(* CoDeSys 2.3.9.41 project: KS Babaevskaya.pro *)
(* Libraries: PID_Regulators.lib 28.12.06 17:47:54, SysLibTime.lib 20.2.06 13:31:16, Util.lib 18.5.10 15:14:28, STANDARD.LIB 4.10.05 11:14:46, IECSFC.LIB 13.4.06 15:51:28, ANALYZATION.LIB 5.10.99 09:05:06 *)

(* PLC configuration (modules and I/O channels)
Fast discrete inputs [I_SIMPLE_INPUT] node 0, in %IB0 out %QB0 {Filtrationtime = 10}
  DD1_DI0 AT %IX0.0 [BitInput] резерв
  DD1_DI1 AT %IX0.1 [BitInput] резерв
  DD1_DI2 AT %IX0.2 [BitInput] резерв
  DD1_DI3 AT %IX0.3 [BitInput] резерв
Discrete inputs [ID130] node 1, in %IB1 out %QB1 {Filtrationtime_GeneralINP = 10; Visibility = No; PinCount = 12}
  AT %IB1.0 [ByteInput] 8 discrete inputs
  AT %IB1.1 [ByteInput] 4 discrete inputs
Discrete outputs [ID131] node 2, in %IB2 out %QB2 {SafeValueByte = 0; SafeValueByteM = 0; Visibility = No; PinCount = 12}
  AT %QB2.0 [ByteOutput] 8 discrete outputs
  AT %QB2.1 [ByteOutput] 4 discrete outputs
ID125	50Hz 2Por	50Hz 2PorBYTEFast analog i AT %IR3.0 [FloatInputP] putsIB%QB%MB%	MDD1_AI0&AI #1 - датчик температуры в помещении {AIN_TYPE = 4-20 mA; Peak_Filtr = 200; Flt_Ch = Off; TauRC = 10; MinFV = 0; MaxFV = 100}
DD1_AI1 AT %IR3.1 [FloatInputP] AI #2 - расходомер FT01.01 (на входе, до отстойника) {AIN_TYPE = 4-20 mA; Peak_Filtr = 200; Flt_Ch = Off; TauRC = 10; MinFV = 0; MaxFV = 600}
DD1_AI2 AT %IR3.2 [FloatInputP] AI #3 - расходомер FT01.02 (на выходе, после отстойника) {AIN_TYPE = 4-20 mA; Peak_Filtr = 200; Flt_Ch = Off; TauRC = 10; MinFV = 0; MaxFV = 600}
DD1_AI3 AT %IR3.3 [FloatInputP] AI #4 - рН-метр QE01.01 (на входе, до отстойника) {AIN_TYPE = 4-20 mA; Peak_Filtr = 200; Flt_Ch = Off; TauRC = 10; MinFV = 0; MaxFV = 20000.0}
DD1_AI4 AT %IR3.4 [FloatInputP] AI #5 - рН-метр QE01.02 (на выходе, после отстойника) {AIN_TYPE = 4-20 mA; Peak_Filtr = 200; Flt_Ch = Off; TauRC = 10; MinFV = 0; MaxFV = 20000.0}
DD1_AI5 AT %IR3.5 [FloatInputP] AI #6 - сигнал от ФПК, давление на входе {AIN_TYPE = 4-20 mA; Peak_Filtr = 200; Flt_Ch = Off; TauRC = 10; MinFV = 0; MaxFV = 20000.0}
DD1_AI6 AT %IR3.6 [FloatInputP] AI #7 - резерв {AIN_TYPE = 4-20 mA; Peak_Filtr = 200; Flt_Ch = Off; TauRC = 10; MinFV = 0; MaxFV = 20000.0}
DD1_AI7 AT %IR3.7 [FloatInputP] AI #8 - обратная связь от ЧРП Н01.05 (частота, обороты, или ток) {AIN_TYPE = 4-20 mA; Peak_Filtr = 200; Flt_Ch = Off; TauRC = 10; MinFV = 0; MaxFV = 20000.0}
AT %IW3.8 [WordInput] AI read time (10ms)
Analog outputs [ID126] node 4, in %IB4 out %QB4
  DD1_AO0 AT %QR4.0 [FloatOutputP] AO #1 - управление ЧРП Н01.05 (поддержание расхода по расходомеру FT01.02) {AOUT_TYPE = 4-20 mA; SafeValueREAL = 0.0}
  DD1_AO1 AT %QR4.1 [FloatOutputP] AO #2 - управление ЧРП НД08.03/01 (подача флокулянта на входе, до отстойника, по FT01.01) {AOUT_TYPE = 4-20 mA; SafeValueREAL = 0.0}
  DD1_AO2 AT %QR4.2 [FloatOutputP] AO #3 - управление ЧРП НД08.03/02 (подача флокулянта на входе, до отстойника, по FT01.01) {AOUT_TYPE = 4-20 mA; SafeValueREAL = 0.0}
  DD1_AO3 AT %QR4.3 [FloatOutputP] AO #4 - управление НД05.02/01 (подача 10%NaCl из УПГ на входе, до отстойника, по FT01.01) {AOUT_TYPE = 4-20 mA; SafeValueREAL = 0.0}
Special input [ID103] node 5, in %IB5 out %QB5 {Filtrationtime = 1000; PinCount = 1; WatchDogPeriod = 400; PollPeriod = 3000; Visibility = No}
  AT %IX5.0 [BitInput] Special input
Special output [ID104] node 6, in %IB6 out %QB6 {Visibility = No; PinCount = 1}
  AT %QX6.0 [BitOutput] Special output
AT %QD7.0 [DWordOutput] Last address
AT %QW7.1 [WordOutput] Last error
RS-485-1 [COM1_USART] node 0, in %IB7.0 out %QB7.0 {CommunicationSpeed = 57600; Parity = NO PARITY CHECK; BitLength = 8 bits; StopLength = One stop bit; InterfaceType = RS485; FrameOriented = RTU; Timeout = 0; Visibility = No}
Universal Modbus device [ID2000] node 1, in %IB7.1 out %QB7.1 {ModuleIP = 10:0:0:102; ServiceTimeout = 20; TCPport = 502; NetMode = Serial; ModuleSlaveAddress = 2; RequestType = Both; PeriodOfService = 100; Visibility = No; RepeatCounter = 0; ByteSequence = Trace_mode}
  AT %QB7.1.0 [ComChannel] Command (0xff - Start)
DD2_DO AT %QD7.1.0.0 [DWordOutput] регистр 0, команда 0х0f
Universal Modbus device [ID2000] node 2, in %IB7.2 out %QB7.2 {ModuleIP = 10:0:0:103; ServiceTimeout = 20; TCPport = 502; NetMode = Serial; ModuleSlaveAddress = 3; RequestType = Both; PeriodOfService = 100; Visibility = No; RepeatCounter = 0; ByteSequence = Trace_mode}
  AT %QB7.2.0 [ComChannel] Command (0xff - Start)
DD3_DO AT %QD7.2.0.0 [DWordOutput]
Universal Modbus device [ID2000] node 3, in %IB7.3 out %QB7.3 {ModuleIP = 10:0:0:104; ServiceTimeout = 20; TCPport = 502; NetMode = Serial; ModuleSlaveAddress = 4; RequestType = Both; PeriodOfService = 100; Visibility = No; RepeatCounter = 0; ByteSequence = Trace_mode}
  AT %QB7.3.0 [ComChannel] Command (0xff - Start)
DD4_DO AT %QD7.3.0.0 [DWordOutput]
Universal Modbus device [ID2000] node 4, in %IB7.4 out %QB7.4 {ModuleIP = 10:0:0:105; ServiceTimeout = 20; TCPport = 502; NetMode = Serial; ModuleSlaveAddress = 5; RequestType = Both; PeriodOfService = 100; Visibility = No; RepeatCounter = 0; ByteSequence = Trace_mode}
  AT %QB7.4.0 [ComChannel] Command (0xff - Start)
DD5_DI AT %ID7.4.0.0 [DWordInput]
Universal Modbus device [ID2000] node 5, in %IB7.5 out %QB7.5 {ModuleIP = 10:0:0:106; ServiceTimeout = 20; TCPport = 502; NetMode = Serial; ModuleSlaveAddress = 6; RequestType = Both; PeriodOfService = 100; Visibility = No; RepeatCounter = 0; ByteSequence = Trace_mode}
  AT %QB7.5.0 [ComChannel] Command (0xff - Start)
DD6_DI AT %ID7.5.0.0 [DWordInput]
Universal Modbus device [ID2000] node 6, in %IB7.6 out %QB7.6 {ModuleIP = 10:0:0:107; ServiceTimeout = 20; TCPport = 502; NetMode = Serial; ModuleSlaveAddress = 7; RequestType = Both; PeriodOfService = 100; Visibility = No; RepeatCounter = 0; ByteSequence = Trace_mode}
  AT %QB7.6.0 [ComChannel] Command (0xff - Start)
DD7_DI AT %ID7.6.0.0 [DWordInput]
Universal Modbus device [ID2000] node 7, in %IB7.7 out %QB7.7 {ModuleIP = 10:0:0:108; ServiceTimeout = 20; TCPport = 502; NetMode = Serial; ModuleSlaveAddress = 8; RequestType = Both; PeriodOfService = 100; Visibility = No; RepeatCounter = 0; ByteSequence = Trace_mode}
  AT %QB7.7.0 [ComChannel] Command (0xff - Start)
DD8_DI AT %ID7.7.0.0 [DWordInput]
Universal Modbus device [ID2000] node 8, in %IB7.8 out %QB7.8 {ModuleIP = 10:0:0:109; ServiceTimeout = 20; TCPport = 502; NetMode = Serial; ModuleSlaveAddress = 9; RequestType = Both; PeriodOfService = 100; Visibility = No; RepeatCounter = 0; ByteSequence = Trace_mode}
  AT %QB7.8.0 [ComChannel] Command (0xff - Start)
DD9_DI AT %ID7.8.0.0 [DWordInput]
Universal Modbus device [ID2000] node 9, in %IB7.9 out %QB7.9 {ModuleIP = 10:0:0:110; ServiceTimeout = 20; TCPport = 502; NetMode = Serial; ModuleSlaveAddress = 10; RequestType = Both; PeriodOfService = 100; Visibility = No; RepeatCounter = 0; ByteSequence = Trace_mode}
  AT %QB7.9.0 [ComChannel] Command (0xff - Start)
DD10_AO0 AT %QW7.9.0.0 [WordOutput]
DD10_AO1 AT %QW7.9.1.0 [WordOutput]
DD10_AO2 AT %QW7.9.2.0 [WordOutput]
DD10_AO3 AT %QW7.9.3.0 [WordOutput]
DD10_AO4 AT %QW7.9.4.0 [WordOutput]
DD10_AO5 AT %QW7.9.5.0 [WordOutput]
DD10_AO6 AT %QW7.9.6.0 [WordOutput]
DD10_AO7 AT %QW7.9.7.0 [WordOutput]
*)

(* POU PLC_PRG, CFC *)
PROGRAM PLC_PRG
VAR
	temperatureLimits: LIMITALARM;		(*блок контроля границ допустимой температуры в помещении*)
	minTemperature: BYTE;		(*температура, ниже которой будет подан сигнал НИЗКАЯ ТЕМПЕРАТУРА*)
	maxTemperature: BYTE;		(*Температура, выше которой будет подан сигнал ВЫСОКАЯ ТЕМПЕРАТУРА*)
	alarmHighTemperature: BOOL;		(*температура выше заданного диапазона*)
	alarmLowTemperature: BOOL;		(*температура ниже заданного диапазона*)
	temperatureValue: REAL;		(*значение температуры в помещении*)
	DD1_AI0_temperature: DECODE_FLOAT;		(*блок контроля состояния аналогового входа ПЛК для датчика температуры в помещении*)
	DD1_AI1_flow: DECODE_FLOAT;		(*блок контроля состояния аналогового входа ПЛК для расходомера FT01.01*)
	DD1_AI1_error: BOOL;		(*авария входа AI2 (возможно, обрыв)*)
	DD1_AI0_error: BOOL;		(*авария входа AI1 (возможно, обрыв)*)


	tempCTU1: CTU;
	tempStartAuto: BOOL;
	tempReset1: BOOL;
	tempReset2: BOOL;
	tempPV: WORD := 15;		(*по умолчанию = 15*)
	tempCTU2: CTU;
	tempStartPump1: BOOL;
	tempStartPump2: BOOL;
	counterPump1: WORD;
	counterPump2: WORD;
	tempErrorPump1: BOOL;
	tempErrorPump2: BOOL;
	tempStopPump1: BOOL;
	tempStopPump2: BOOL;
	tempFtrigPump1: F_TRIG;
	tempRtrigPump1: R_TRIG;
	tempRSpump1: RS;
	tempStartStopPump1: BOOL;
	tempStartStopPump2: BOOL;
	tempPump1ON: BOOL;
	tempPump2ON: BOOL;
	tempRtrigPump2: R_TRIG;
	tempFtrigPump2: F_TRIG;
	tempRSpump2: RS;
	errorPump1Trig: RS;
	tempAlarmReset: BOOL;
	errorPump2Trig: RS;
	tempPump1EmergencyON: BOOL;
	tempPump1NormalON: BOOL;
	tempPump2NormalON: BOOL;
	tempPump2EmergencyON: BOOL;
	tempMan2Pump: ManualTwoPumpManager;
	tempalarmPump1: BOOL;
	tempalarmPump2: BOOL;
	tempalarmPump1RStrig: RS;
	tempalarmPump2RStrig: RS;
	alarmReset: BOOL;
	startStopPump1: BOOL;
	pump2ON: BOOL;
	alarmPump1: BOOL;
	startStopPump2: BOOL;
	pump1ON: BOOL;
	alarmPump2: BOOL;
	alarmPump2RStrig: RS;
	pump1EmergencyON: BOOL;
	pump2NormalON: BOOL;
	pump2EmergencyON: BOOL;
	RSpump2: RS;
	RtrigPump2: R_TRIG;
	FtrigPump2: F_TRIG;
	alarmPump1RStrig: RS;
	pump1NormalON: BOOL;
	RSpump1: RS;
	FtrigPump1: F_TRIG;
	RtrigPump1: R_TRIG;
	counterStart: BOOL;
	counterPump1ON: BOOL;
	counterPump2ON: BOOL;
	tempRtrig: R_TRIG;
	tempFtrig: F_TRIG;
	tempRStrig: RS;
	tempSRtrig2: SR;
	tempSRtrig1: SR;
	tempRStrig1: RS;
	tempRStrig2: RS;
	tempValueToResetCTU: WORD;
	tempCTU1reset: BOOL;
	tempCTU2reset: BOOL;
	tempCounterStart: BOOL;
	tempCounterPump1: WORD;
	tempCounterPump2: WORD;
	tempCounterTwoPumpManager: CounterTwoPumpManager;
	tempTON1: TON;
	tempBLINK: BLINK;
	tempRTC: RTC;
	tempCTU21: CTU;
	tempTIMEcdt: DT;
	tempTIMEPDT: DT;
	tempCTU22: CTU;
	tempSema1: SEMA;
	tempFTrig21: F_TRIG;
	tempTIME: TIME;
	tempTimeBlink: TIME;
	tempTIMEboolQ: BOOL;
	workTimePump1ON: BOOL;
	workTimePump2ON: BOOL;
	tempTIME2: TIME;
	tempRTrig23: R_TRIG;
	tempRStrig24: RS;
	tempRStrigTIME2: RS;
	tempRStrigTIME: RS;
	tempTOF1: TOF;
	tempTP1: TP;
	tempRStrig23: RS;
	tempRTrig21: R_TRIG;
	tempVARtime: DWORD;
	tempRStrig11: RS;
	tempRStrig12: RS;
	tempFtrig22: F_TRIG;
	tempFTrig24: F_TRIG;
	tempFTrig25: F_TRIG;
	currentWorkTimePump1: TIME;
	currentWorkTimePump2: TIME;
	tempTwoPumpFullManager: TwoPumpManager;
	tempWorkTimeStart: BOOL;
	pump1Time: TIME;
	pump2Time: TIME;
	tempWorkTimeReset: BOOL;
END_VAR
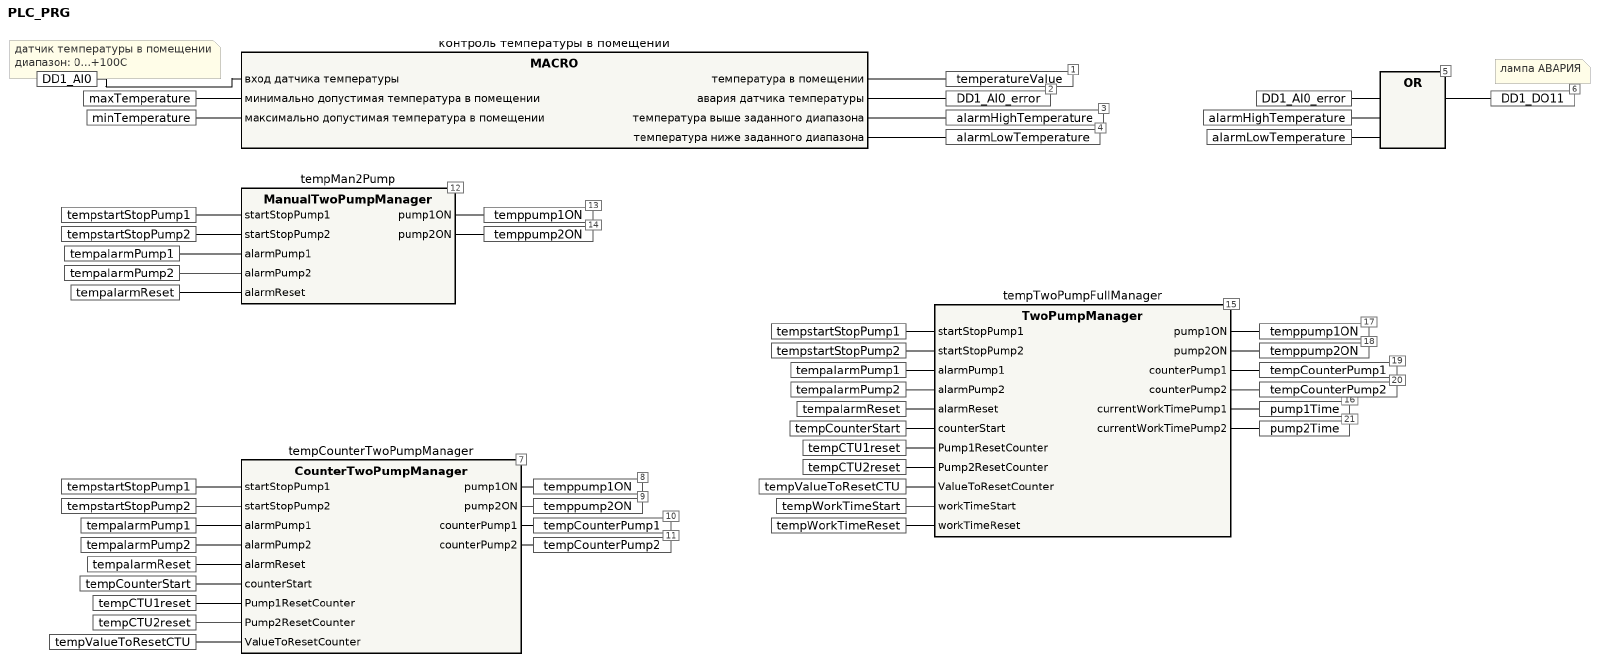
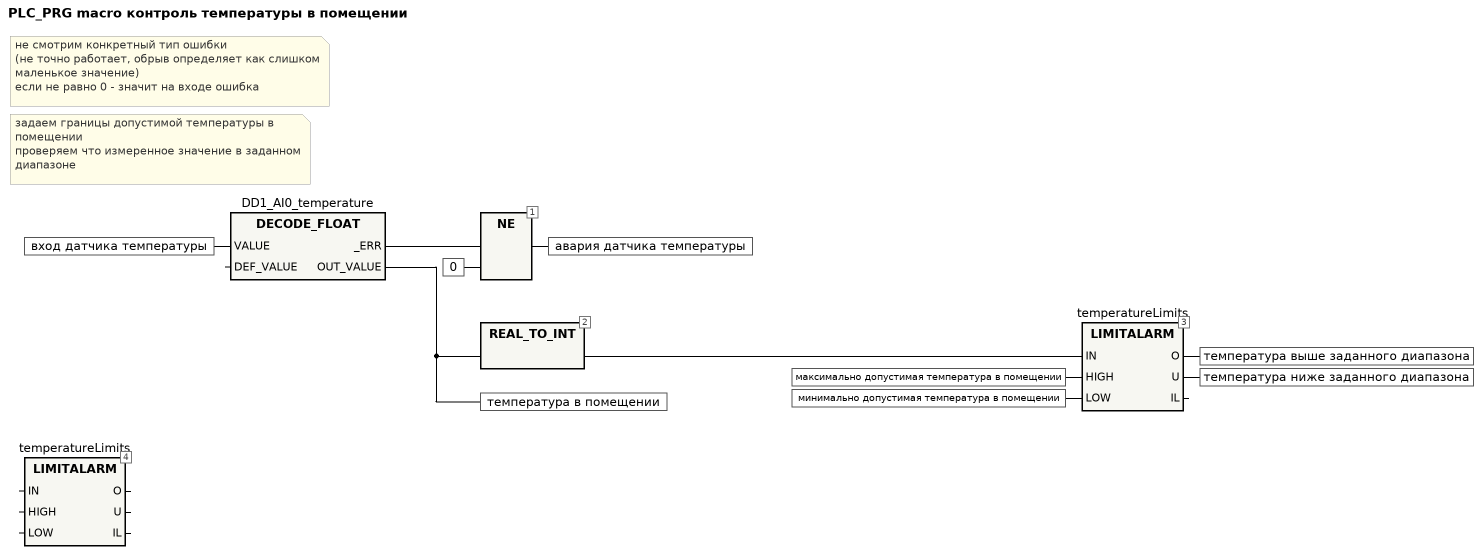
_CFC_ (* Continuous Function Chart, elements in execution order *)
(* датчик температуры в помещении / диапазон: 0...+100С *)
(* лампа АВАРИЯ *)
#0 MACRO контроль температуры в помещении(pin 1 "вход датчика температуры": DD1_AI0, pin 2 "минимально допустимая температура в помещении": maxTemperature, pin 3 "максимально допустимая температура в помещении": minTemperature)
	(* не смотрим конкретный тип ошибки / (не точно работает, обрыв определяет как слишком маленькое значение) / если не равно 0 - значит на входе ошибка *)
	(* задаем границы допустимой температуры в помещении / проверяем что измеренное значение в заданном диапазоне *)
	#1 DD1_AI0_temperature:DECODE_FLOAT(VALUE: pin 1, DEF_VALUE: -)
	#2 NE(#1._ERR, 0)
	out 2 "авария датчика температуры" <= #2
	out 1 "температура в помещении" <= #1.OUT_VALUE
	#3 REAL_TO_INT(#1.OUT_VALUE)
	#4 temperatureLimits:LIMITALARM(IN: #3, HIGH: pin 3, LOW: pin 2)
	out 3 "температура выше заданного диапазона" <= #4.O
	out 4 "температура ниже заданного диапазона" <= #4.U
	#5 temperatureLimits:LIMITALARM(IN: -, HIGH: -, LOW: -)
END_MACRO
#6 temperatureValue <= #0.out 1
#7 DD1_AI0_error <= #0.out 2
#8 alarmHighTemperature <= #0.out 3
#9 alarmLowTemperature <= #0.out 4
#10 OR(DD1_AI0_error, alarmHighTemperature, alarmLowTemperature)
#11 DD1_DO11 <= #10
#12 tempCounterTwoPumpManager:CounterTwoPumpManager(startStopPump1: tempstartStopPump1, startStopPump2: tempstartStopPump2, alarmPump1: tempalarmPump1, alarmPump2: tempalarmPump2, alarmReset: tempalarmReset, counterStart: tempCounterStart, Pump1ResetCounter: tempCTU1reset, Pump2ResetCounter: tempCTU2reset, ValueToResetCounter: tempValueToResetCTU)
#13 temppump1ON <= #12.pump1ON
#14 temppump2ON <= #12.pump2ON
#15 tempCounterPump1 <= #12.counterPump1
#16 tempCounterPump2 <= #12.counterPump2
#17 tempMan2Pump:ManualTwoPumpManager(startStopPump1: tempstartStopPump1, startStopPump2: tempstartStopPump2, alarmPump1: tempalarmPump1, alarmPump2: tempalarmPump2, alarmReset: tempalarmReset)
#18 temppump1ON <= #17.pump1ON
#19 temppump2ON <= #17.pump2ON
#20 tempTwoPumpFullManager:TwoPumpManager(startStopPump1: tempstartStopPump1, startStopPump2: tempstartStopPump2, alarmPump1: tempalarmPump1, alarmPump2: tempalarmPump2, alarmReset: tempalarmReset, counterStart: tempCounterStart, Pump1ResetCounter: tempCTU1reset, Pump2ResetCounter: tempCTU2reset, ValueToResetCounter: tempValueToResetCTU, workTimeStart: tempWorkTimeStart, workTimeReset: tempWorkTimeReset)
#21 pump1Time <= #20.currentWorkTimePump1
#22 temppump1ON <= #20.pump1ON
#23 temppump2ON <= #20.pump2ON
#24 tempCounterPump1 <= #20.counterPump1
#25 tempCounterPump2 <= #20.counterPump2
#26 pump2Time <= #20.currentWorkTimePump2
_END_CFC_
(* the same logic as Structured Text *)
(* датчик температуры в помещении / диапазон: 0...+100С *)
(* лампа АВАРИЯ *)
(* macro контроль температуры в помещении *)
(* не смотрим конкретный тип ошибки / (не точно работает, обрыв определяет как слишком маленькое значение) / если не равно 0 - значит на входе ошибка *)
(* задаем границы допустимой температуры в помещении / проверяем что измеренное значение в заданном диапазоне *)
DD1_AI0_temperature(VALUE := DD1_AI0);
temperatureLimits(IN := REAL_TO_INT(DD1_AI0_temperature.OUT_VALUE), HIGH := minTemperature, LOW := maxTemperature);
temperatureLimits();
temperatureValue := DD1_AI0_temperature.OUT_VALUE;
DD1_AI0_error := DD1_AI0_temperature._ERR <> 0;
alarmHighTemperature := temperatureLimits.O;
alarmLowTemperature := temperatureLimits.U;
DD1_DO11 := DD1_AI0_error OR alarmHighTemperature OR alarmLowTemperature;
tempCounterTwoPumpManager(startStopPump1 := tempstartStopPump1, startStopPump2 := tempstartStopPump2, alarmPump1 := tempalarmPump1, alarmPump2 := tempalarmPump2, alarmReset := tempalarmReset, counterStart := tempCounterStart, Pump1ResetCounter := tempCTU1reset, Pump2ResetCounter := tempCTU2reset, ValueToResetCounter := tempValueToResetCTU);
temppump1ON := tempCounterTwoPumpManager.pump1ON;
temppump2ON := tempCounterTwoPumpManager.pump2ON;
tempCounterPump1 := tempCounterTwoPumpManager.counterPump1;
tempCounterPump2 := tempCounterTwoPumpManager.counterPump2;
tempMan2Pump(startStopPump1 := tempstartStopPump1, startStopPump2 := tempstartStopPump2, alarmPump1 := tempalarmPump1, alarmPump2 := tempalarmPump2, alarmReset := tempalarmReset);
temppump1ON := tempMan2Pump.pump1ON;
temppump2ON := tempMan2Pump.pump2ON;
tempTwoPumpFullManager(startStopPump1 := tempstartStopPump1, startStopPump2 := tempstartStopPump2, alarmPump1 := tempalarmPump1, alarmPump2 := tempalarmPump2, alarmReset := tempalarmReset, counterStart := tempCounterStart, Pump1ResetCounter := tempCTU1reset, Pump2ResetCounter := tempCTU2reset, ValueToResetCounter := tempValueToResetCTU, workTimeStart := tempWorkTimeStart, workTimeReset := tempWorkTimeReset);
pump1Time := tempTwoPumpFullManager.currentWorkTimePump1;
temppump1ON := tempTwoPumpFullManager.pump1ON;
temppump2ON := tempTwoPumpFullManager.pump2ON;
tempCounterPump1 := tempTwoPumpFullManager.counterPump1;
tempCounterPump2 := tempTwoPumpFullManager.counterPump2;
pump2Time := tempTwoPumpFullManager.currentWorkTimePump2;
END_PROGRAM

(* POU ManualTwoPumpManager, CFC *)
FUNCTION_BLOCK ManualTwoPumpManager
VAR_INPUT
	startStopPump1: BOOL;		(*Сигнал на пуск/стоп первого насоса.*)
	startStopPump2: BOOL;		(*Сигнал на пуск/стоп второго насоса.*)
	alarmPump1: BOOL;		(*Сигнал "авария" на первом насосе.*)
	alarmPump2: BOOL;		(*Сигнал "авария" на втором насосе.*)
	alarmReset: BOOL;		(*Сброс аварии.*)
END_VAR
VAR_OUTPUT
	pump1ON: BOOL;		(*Выход на включение первого насоса.*)
	pump2ON: BOOL;		(*Выход на включение второго насоса.*)
END_VAR
VAR
	RtrigPump1: R_TRIG;		(*Включает первый насос по фронту сигнала на ручной пуск/стоп.*)
	FtrigPump1: F_TRIG;		(*Выключает первый насос по спаду сигнала на ручной пуск/стоп.*)
	RtrigPump2: R_TRIG;		(*Включает второй насос по фронту сигнала на ручной пуск/стоп.*)
	FtrigPump2: F_TRIG;		(*Выключает второй насос по спаду сигнала на ручной пуск/стоп.*)
	RSpump1: RS;		(*RS-триггер нормального включения первого насоса*)
	RSpump2: RS;		(*RS-триггер нормального включения второго насоса*)
	pump1NormalON: BOOL;		(*Сигнал нормального (неаварийного) включения первого насоса.*)
	pump2NormalON: BOOL;		(*Сигнал нормального (неаварийного) включения второго насоса.*)
	pump2EmergencyON: BOOL;		(*Сигнал аварийного включения второго насоса (при аварии первого).*)
	pump1EmergencyON: BOOL;		(*Сигнал аварийного включения первого насоса (при аварии второго).*)
	alarmPump1RStrig: RS;		(*Триггер аварии первого насоса.*)
	alarmPump2RStrig: RS;		(*Триггер аварии второго насоса.*)
END_VAR
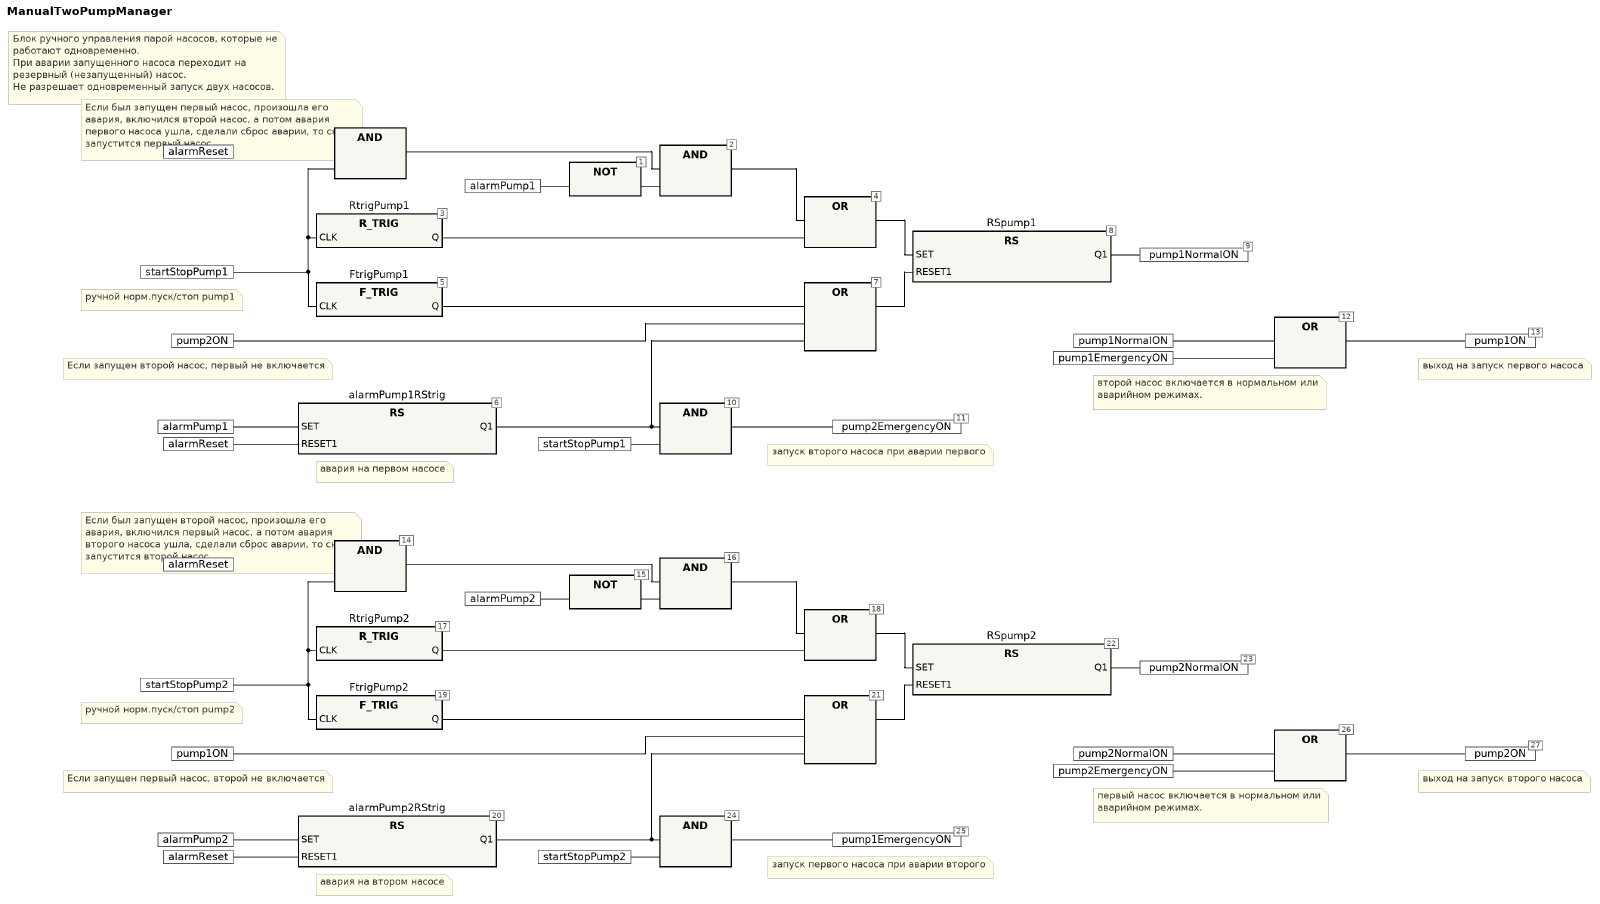
_CFC_ (* Continuous Function Chart, elements in execution order *)
(* выход на запуск второго насоса *)
(* запуск первого насоса при аварии второго *)
(* Если запущен первый насос, второй не включается *)
(* авария на втором насосе *)
(* ручной норм.пуск/стоп pump2 *)
(* выход на запуск первого насоса *)
(* ручной норм.пуск/стоп pump1 *)
(* запуск второго насоса при аварии первого *)
(* Если запущен второй насос, первый не включается *)
(* авария на первом насосе *)
(* Блок ручного управления парой насосов, которые не работают одновременно. / При аварии запущенного насоса переходит на резервный (незапущенный) насос. / Не разрешает одновременный запуск двух насосов. *)
(* Если был запущен первый насос, произошла его авария, включился второй насос, а потом авария первого насоса ушла, сделали сброс аварии, то снова запустится первый насос. *)
(* второй насос включается в нормальном или аварийном режимах. *)
(* первый насос включается в нормальном или аварийном режимах. *)
(* Если был запущен второй насос, произошла его авария, включился первый насос, а потом авария второго насоса ушла, сделали сброс аварии, то снова запустится второй насос. *)
#0 AND(alarmReset, startStopPump1)
#1 NOT(alarmPump1)
#2 AND(#0, #1)
#3 RtrigPump1:R_TRIG(CLK: startStopPump1)
#4 OR(#2, #3.Q)
#5 FtrigPump1:F_TRIG(CLK: startStopPump1)
#6 alarmPump1RStrig:RS(SET: alarmPump1, RESET1: alarmReset)
#7 OR(#5.Q, pump2ON, #6.Q1)
#8 RSpump1:RS(SET: #4, RESET1: #7)
#9 pump1NormalON <= #8.Q1
#10 AND(#6.Q1, startStopPump1)
#11 pump2EmergencyON <= #10
#12 OR(pump1NormalON, pump1EmergencyON)
#13 pump1ON <= #12
#14 AND(alarmReset, startStopPump2)
#15 NOT(alarmPump2)
#16 AND(#14, #15)
#17 RtrigPump2:R_TRIG(CLK: startStopPump2)
#18 OR(#16, #17.Q)
#19 FtrigPump2:F_TRIG(CLK: startStopPump2)
#20 alarmPump2RStrig:RS(SET: alarmPump2, RESET1: alarmReset)
#21 OR(#19.Q, pump1ON, #20.Q1)
#22 RSpump2:RS(SET: #18, RESET1: #21)
#23 pump2NormalON <= #22.Q1
#24 AND(#20.Q1, startStopPump2)
#25 pump1EmergencyON <= #24
#26 OR(pump2NormalON, pump2EmergencyON)
#27 pump2ON <= #26
_END_CFC_
(* the same logic as Structured Text *)
(* выход на запуск второго насоса *)
(* запуск первого насоса при аварии второго *)
(* Если запущен первый насос, второй не включается *)
(* авария на втором насосе *)
(* ручной норм.пуск/стоп pump2 *)
(* выход на запуск первого насоса *)
(* ручной норм.пуск/стоп pump1 *)
(* запуск второго насоса при аварии первого *)
(* Если запущен второй насос, первый не включается *)
(* авария на первом насосе *)
(* Блок ручного управления парой насосов, которые не работают одновременно. / При аварии запущенного насоса переходит на резервный (незапущенный) насос. / Не разрешает одновременный запуск двух насосов. *)
(* Если был запущен первый насос, произошла его авария, включился второй насос, а потом авария первого насоса ушла, сделали сброс аварии, то снова запустится первый насос. *)
(* второй насос включается в нормальном или аварийном режимах. *)
(* первый насос включается в нормальном или аварийном режимах. *)
(* Если был запущен второй насос, произошла его авария, включился первый насос, а потом авария второго насоса ушла, сделали сброс аварии, то снова запустится второй насос. *)
RtrigPump1(CLK := startStopPump1);
FtrigPump1(CLK := startStopPump1);
alarmPump1RStrig(SET := alarmPump1, RESET1 := alarmReset);
RSpump1(SET := ((alarmReset AND startStopPump1) AND NOT alarmPump1) OR RtrigPump1.Q, RESET1 := FtrigPump1.Q OR pump2ON OR alarmPump1RStrig.Q1);
pump1NormalON := RSpump1.Q1;
pump2EmergencyON := alarmPump1RStrig.Q1 AND startStopPump1;
pump1ON := pump1NormalON OR pump1EmergencyON;
RtrigPump2(CLK := startStopPump2);
FtrigPump2(CLK := startStopPump2);
alarmPump2RStrig(SET := alarmPump2, RESET1 := alarmReset);
RSpump2(SET := ((alarmReset AND startStopPump2) AND NOT alarmPump2) OR RtrigPump2.Q, RESET1 := FtrigPump2.Q OR pump1ON OR alarmPump2RStrig.Q1);
pump2NormalON := RSpump2.Q1;
pump1EmergencyON := alarmPump2RStrig.Q1 AND startStopPump2;
pump2ON := pump2NormalON OR pump2EmergencyON;
END_FUNCTION_BLOCK

(* POU CounterTwoPumpManager, CFC *)
FUNCTION_BLOCK CounterTwoPumpManager
VAR_INPUT
	startStopPump1: BOOL;		(*Сигнал на пуск/стоп первого насоса.*)
	startStopPump2: BOOL;		(*Сигнал на пуск/стоп второго насоса.*)
	alarmPump1: BOOL;		(*Сигнал "авария" на первом насосе.*)
	alarmPump2: BOOL;		(*Сигнал "авария" на втором насосе.*)
	alarmReset: BOOL;		(*Сброс аварии.*)

	counterStart: BOOL;		(*Запуск насоса с меньшим количеством включений.*)
	Pump1ResetCounter: BOOL;		(*Сброс счетчика количества включений первого насоса. Сбрасывается также автоматически при достижении счетчиком значения ValueToResetCTU.*)
	Pump2ResetCounter: BOOL;		(*Сброс счетчика количества включений второго насоса. Сбрасывается также автоматически при достижении счетчиком значения ValueToResetCTU.*)
	ValueToResetCounter: WORD := 65535;		(*Значение счетчика, после которого он сбрасывается на ноль. Максимальное допустимое значение: 65535, оно же установлено по умолчанию, сработает, если не подключать ко входу переменную.*)
END_VAR
VAR_OUTPUT
	pump1ON: BOOL;		(*Выход на включение первого насоса.*)
	pump2ON: BOOL;		(*Выход на включение второго насоса.*)

	counterPump1: WORD;		(*Количество включений первого насоса. При достижении значения ValueToResetCTU сбрасывается в ноль.*)
	counterPump2: WORD;		(*Количество включений второго насоса. При достижении значения ValueToResetCTU сбрасывается в ноль.*)
END_VAR
VAR
	RtrigPump1: R_TRIG;		(*Включает первый насос по фронту сигнала на ручной пуск/стоп.*)
	FtrigPump1: F_TRIG;		(*Выключает первый насос по спаду сигнала на ручной пуск/стоп.*)
	RtrigPump2: R_TRIG;		(*Включает второй насос по фронту сигнала на ручной пуск/стоп.*)
	FtrigPump2: F_TRIG;		(*Выключает второй насос по спаду сигнала на ручной пуск/стоп.*)
	RSpump1: RS;		(*RS-триггер нормального включения первого насоса*)
	RSpump2: RS;		(*RS-триггер нормального включения второго насоса*)
	pump1NormalON: BOOL;		(*Сигнал нормального (неаварийного) включения первого насоса.*)
	pump2NormalON: BOOL;		(*Сигнал нормального (неаварийного) включения второго насоса.*)
	pump2EmergencyON: BOOL;		(*Сигнал аварийного включения второго насоса (при аварии первого).*)
	pump1EmergencyON: BOOL;		(*Сигнал аварийного включения первого насоса (при аварии второго).*)
	alarmPump1RStrig: RS;		(*Триггер аварии первого насоса.*)
	alarmPump2RStrig: RS;		(*Триггер аварии второго насоса.*)

	CTUPump1: CTU;		(*Счетчик количества включений первого насоса.*)
	CTUPump2: CTU;		(*Счетчик количества включений второго насоса.*)
	counterRtrig: R_TRIG;		(*Детектор переднего фронта сигнала на старт насоса с меньшей наработкой, включает насос.*)
	counterFtrig: F_TRIG;		(*Детектор спада сигнала на запуск насоса с меньшей наработкой, останавливает насос.*)
	counterRStrigPump1: RS;		(*Триггер-защелка включения первого насоса при запуске по количеству включений.*)
	counterRStrigPump2: RS;		(*Триггер-защелка включения второго насоса при запуске по количеству включений.*)
	counterPump1ON: BOOL;		(*Сигнал на запуск первого насоса при запуске по количеству включений.*)
	counterPump2ON: BOOL;		(*Сигнал на запуск второго насоса при запуске по количеству включений.*)
END_VAR
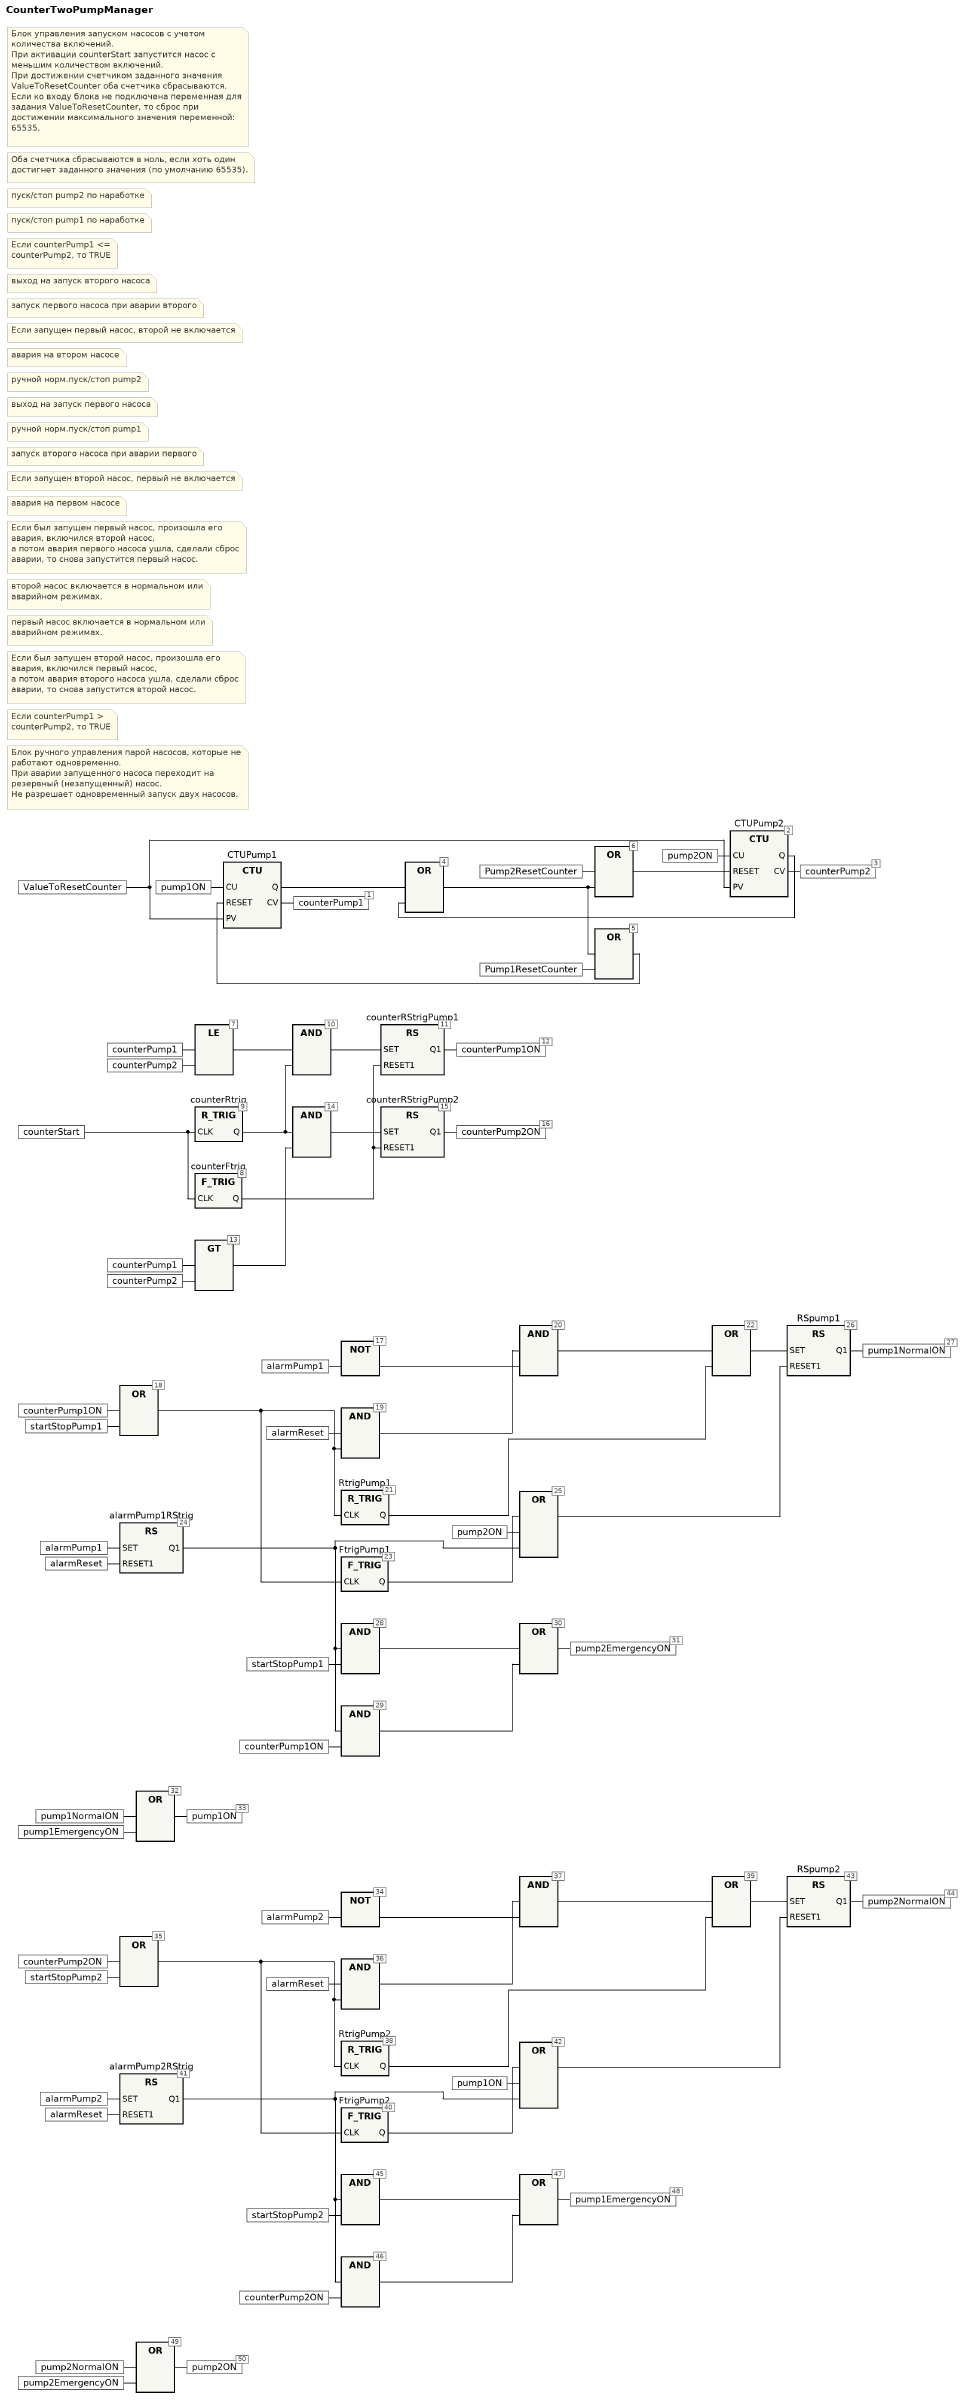
_CFC_ (* Continuous Function Chart, elements in execution order *)
(* Блок управления запуском насосов с учетом количества включений. / При активации counterStart запустится насос с меньшим количеством включений. / При достижении счетчиком заданного значения ValueToResetCounter оба счетчика сбрасываются. / Если ко входу блока не подключена переменная для задания ValueToResetCounter, то сброс при достижении максимального значения переменной: 65535. *)
(* Оба счетчика сбрасываются в ноль, если хоть один достигнет заданного значения (по умолчанию 65535). *)
(* пуск/стоп pump2 по наработке *)
(* пуск/стоп pump1 по наработке *)
(* Если counterPump1 <= / counterPump2, то TRUE *)
(* выход на запуск второго насоса *)
(* запуск первого насоса при аварии второго *)
(* Если запущен первый насос, второй не включается *)
(* авария на втором насосе *)
(* ручной норм.пуск/стоп pump2 *)
(* выход на запуск первого насоса *)
(* ручной норм.пуск/стоп pump1 *)
(* запуск второго насоса при аварии первого *)
(* Если запущен второй насос, первый не включается *)
(* авария на первом насосе *)
(* Если был запущен первый насос, произошла его авария, включился второй насос, / а потом авария первого насоса ушла, сделали сброс аварии, то снова запустится первый насос. *)
(* второй насос включается в нормальном или аварийном режимах. *)
(* первый насос включается в нормальном или аварийном режимах. *)
(* Если был запущен второй насос, произошла его авария, включился первый насос, / а потом авария второго насоса ушла, сделали сброс аварии, то снова запустится второй насос. *)
(* Если counterPump1 > / counterPump2, то TRUE *)
(* Блок ручного управления парой насосов, которые не работают одновременно. / При аварии запущенного насоса переходит на резервный (незапущенный) насос. / Не разрешает одновременный запуск двух насосов. *)
#0 CTUPump1:CTU(CU: pump1ON, RESET: #5, PV: ValueToResetCounter)
#1 counterPump1 <= #0.CV
#2 CTUPump2:CTU(CU: pump2ON, RESET: #6, PV: ValueToResetCounter)
#3 counterPump2 <= #2.CV
#4 OR(#0.Q, #2.Q)
#5 OR(#4, Pump1ResetCounter)
#6 OR(Pump2ResetCounter, #4)
#7 LE(counterPump1, counterPump2)
#8 counterFtrig:F_TRIG(CLK: counterStart)
#9 counterRtrig:R_TRIG(CLK: counterStart)
#10 AND(#7, #9.Q)
#11 counterRStrigPump1:RS(SET: #10, RESET1: #8.Q)
#12 counterPump1ON <= #11.Q1
#13 GT(counterPump1, counterPump2)
#14 AND(#9.Q, #13)
#15 counterRStrigPump2:RS(SET: #14, RESET1: #8.Q)
#16 counterPump2ON <= #15.Q1
#17 NOT(alarmPump1)
#18 OR(counterPump1ON, startStopPump1)
#19 AND(alarmReset, #18)
#20 AND(#19, #17)
#21 RtrigPump1:R_TRIG(CLK: #18)
#22 OR(#20, #21.Q)
#23 FtrigPump1:F_TRIG(CLK: #18)
#24 alarmPump1RStrig:RS(SET: alarmPump1, RESET1: alarmReset)
#25 OR(#23.Q, pump2ON, #24.Q1)
#26 RSpump1:RS(SET: #22, RESET1: #25)
#27 pump1NormalON <= #26.Q1
#28 AND(#24.Q1, startStopPump1)
#29 AND(#24.Q1, counterPump1ON)
#30 OR(#28, #29)
#31 pump2EmergencyON <= #30
#32 OR(pump1NormalON, pump1EmergencyON)
#33 pump1ON <= #32
#34 NOT(alarmPump2)
#35 OR(counterPump2ON, startStopPump2)
#36 AND(alarmReset, #35)
#37 AND(#36, #34)
#38 RtrigPump2:R_TRIG(CLK: #35)
#39 OR(#37, #38.Q)
#40 FtrigPump2:F_TRIG(CLK: #35)
#41 alarmPump2RStrig:RS(SET: alarmPump2, RESET1: alarmReset)
#42 OR(#40.Q, pump1ON, #41.Q1)
#43 RSpump2:RS(SET: #39, RESET1: #42)
#44 pump2NormalON <= #43.Q1
#45 AND(#41.Q1, startStopPump2)
#46 AND(#41.Q1, counterPump2ON)
#47 OR(#45, #46)
#48 pump1EmergencyON <= #47
#49 OR(pump2NormalON, pump2EmergencyON)
#50 pump2ON <= #49
_END_CFC_
END_FUNCTION_BLOCK

(* POU TwoPumpManager, CFC *)
FUNCTION_BLOCK TwoPumpManager
VAR_INPUT
	startStopPump1: BOOL;		(*Сигнал на пуск/стоп первого насоса.*)
	startStopPump2: BOOL;		(*Сигнал на пуск/стоп второго насоса.*)
	alarmPump1: BOOL;		(*Сигнал "авария" на первом насосе.*)
	alarmPump2: BOOL;		(*Сигнал "авария" на втором насосе.*)
	alarmReset: BOOL;		(*Сброс аварии.*)

	counterStart: BOOL;		(*Запуск насоса с меньшим количеством включений.*)
	Pump1ResetCounter: BOOL;		(*Сброс счетчика количества включений первого насоса. Сбрасывается также автоматически при достижении счетчиком значения ValueToResetCTU.*)
	Pump2ResetCounter: BOOL;		(*Сброс счетчика количества включений второго насоса. Сбрасывается также автоматически при достижении счетчиком значения ValueToResetCTU.*)
	ValueToResetCounter: WORD := 65535;		(*Значение счетчика, после которого он сбрасывается на ноль. Максимальное допустимое значение: 65535, оно же установлено по умолчанию, сработает, если не подключать ко входу переменную.*)

	workTimeStart: BOOL;		(*Запуск насоса с выбором по меньшей наработке.*)
	workTimeReset: BOOL;		(*Сброс времени наработки.*)
END_VAR
VAR_OUTPUT
	pump1ON: BOOL;		(*Выход на включение первого насоса.*)
	pump2ON: BOOL;		(*Выход на включение второго насоса.*)

	counterPump1: WORD;		(*Количество включений первого насоса. При достижении значения ValueToResetCTU сбрасывается в ноль.*)
	counterPump2: WORD;		(*Количество включений второго насоса. При достижении значения ValueToResetCTU сбрасывается в ноль.*)

	currentWorkTimePump1: TIME;		(*Текущая наработка первого насоса.*)
	currentWorkTimePump2: TIME;		(*Текущая наработка второго насоса.*)
END_VAR
VAR
	RtrigPump1: R_TRIG;		(*Включает первый насос по фронту сигнала на ручной пуск/стоп.*)
	FtrigPump1: F_TRIG;		(*Выключает первый насос по спаду сигнала на ручной пуск/стоп.*)
	RtrigPump2: R_TRIG;		(*Включает второй насос по фронту сигнала на ручной пуск/стоп.*)
	FtrigPump2: F_TRIG;		(*Выключает второй насос по спаду сигнала на ручной пуск/стоп.*)
	RSpump1: RS;		(*RS-триггер нормального включения первого насоса*)
	RSpump2: RS;		(*RS-триггер нормального включения второго насоса*)
	pump1NormalON: BOOL;		(*Сигнал нормального (неаварийного) включения первого насоса.*)
	pump2NormalON: BOOL;		(*Сигнал нормального (неаварийного) включения второго насоса.*)
	pump2EmergencyON: BOOL;		(*Сигнал аварийного включения второго насоса (при аварии первого).*)
	pump1EmergencyON: BOOL;		(*Сигнал аварийного включения первого насоса (при аварии второго).*)
	alarmPump1RStrig: RS;		(*Триггер аварии первого насоса.*)
	alarmPump2RStrig: RS;		(*Триггер аварии второго насоса.*)

	CTUPump1: CTU;		(*Счетчик количества включений первого насоса.*)
	CTUPump2: CTU;		(*Счетчик количества включений второго насоса.*)
	counterRtrig: R_TRIG;		(*Детектор переднего фронта сигнала на старт насоса с меньшей наработкой, включает насос.*)
	counterFtrig: F_TRIG;		(*Детектор спада сигнала на запуск насоса с меньшей наработкой, останавливает насос.*)
	counterRStrigPump1: RS;		(*Триггер-защелка включения первого насоса при запуске по количеству включений.*)
	counterRStrigPump2: RS;		(*Триггер-защелка включения второго насоса при запуске по количеству включений.*)
	counterPump1ON: BOOL;		(*Сигнал на запуск первого насоса при запуске по количеству включений.*)
	counterPump2ON: BOOL;		(*Сигнал на запуск второго насоса при запуске по количеству включений.*)

	workTimePump1ON: BOOL;		(*Сигнал на запуск первого насоса при запуске по наработке.*)
	workTimePump2ON: BOOL;		(*Сигнал на запуск второго насоса при запуске по наработке.*)
	timerFtrig: F_TRIG;		(*Детектор спада сигнала работы насосов для записи времени работы.*)
	pump1Ftrig: F_TRIG;		(*Детектор спада сигнала работы первого насоса для подсчета наработки.*)
	pump2Ftrig: F_TRIG;		(*Детектор спада сигнала работы второго насоса для подсчета наработки.*)
	timeStartFtrig: F_TRIG;		(*Детектор спада сигнала на запуск по наработке.*)
	timeStartRtrig: R_TRIG;		(*Детектор переднего фронта сигнала на запуск по наработке.*)
	timerRTC: RTC;		(*Таймер реального времени для подсчета наработки.*)
	timeCDT: DT;		(*Время на выходе таймера реального времени.*)
	timePDT: DT;		(*Время на входе таймера реального времени. Не инициализируется, чтобы подсчет всегда начинался от нуля.*)
	tempVarTime: TIME;		(*Промежуточная переменная хранения времени наработки за включение.*)
	workTimePump1: TIME;		(*Время наработки первого насоса. Подсчитывается после выключения насоса.*)
	workTimePump2: TIME;		(*Время наработки второго насоса. Подсчитывается после выключения насоса.*)
	RStrigTimePump1: RS;		(*Триггер-защелка запуск первого насоса по наработке.*)
	RStrigTimePump2: RS;		(*Триггер-защелка запуск второго насоса по наработке.*)
END_VAR
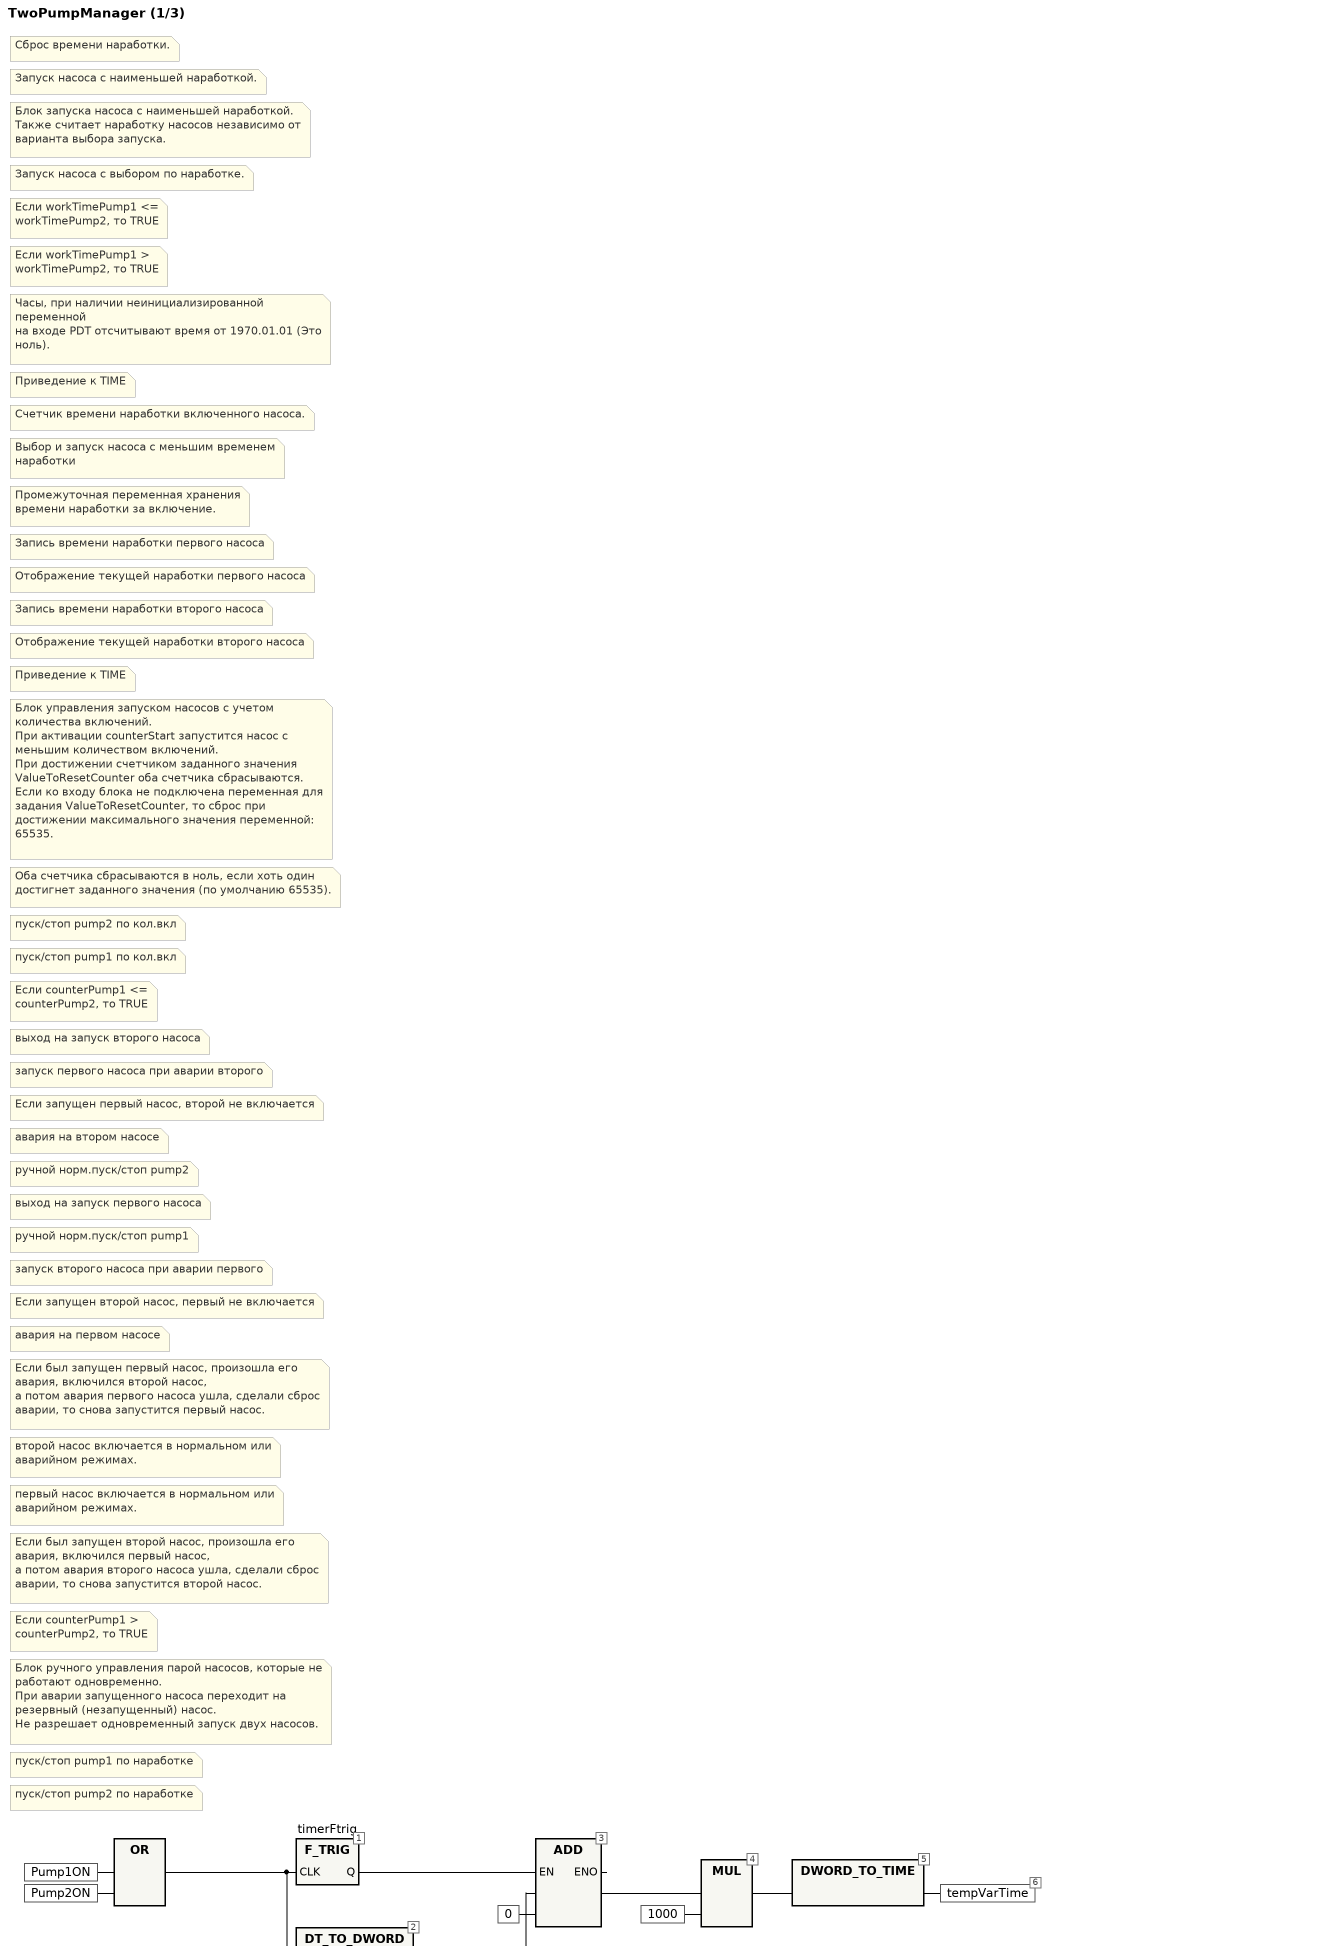
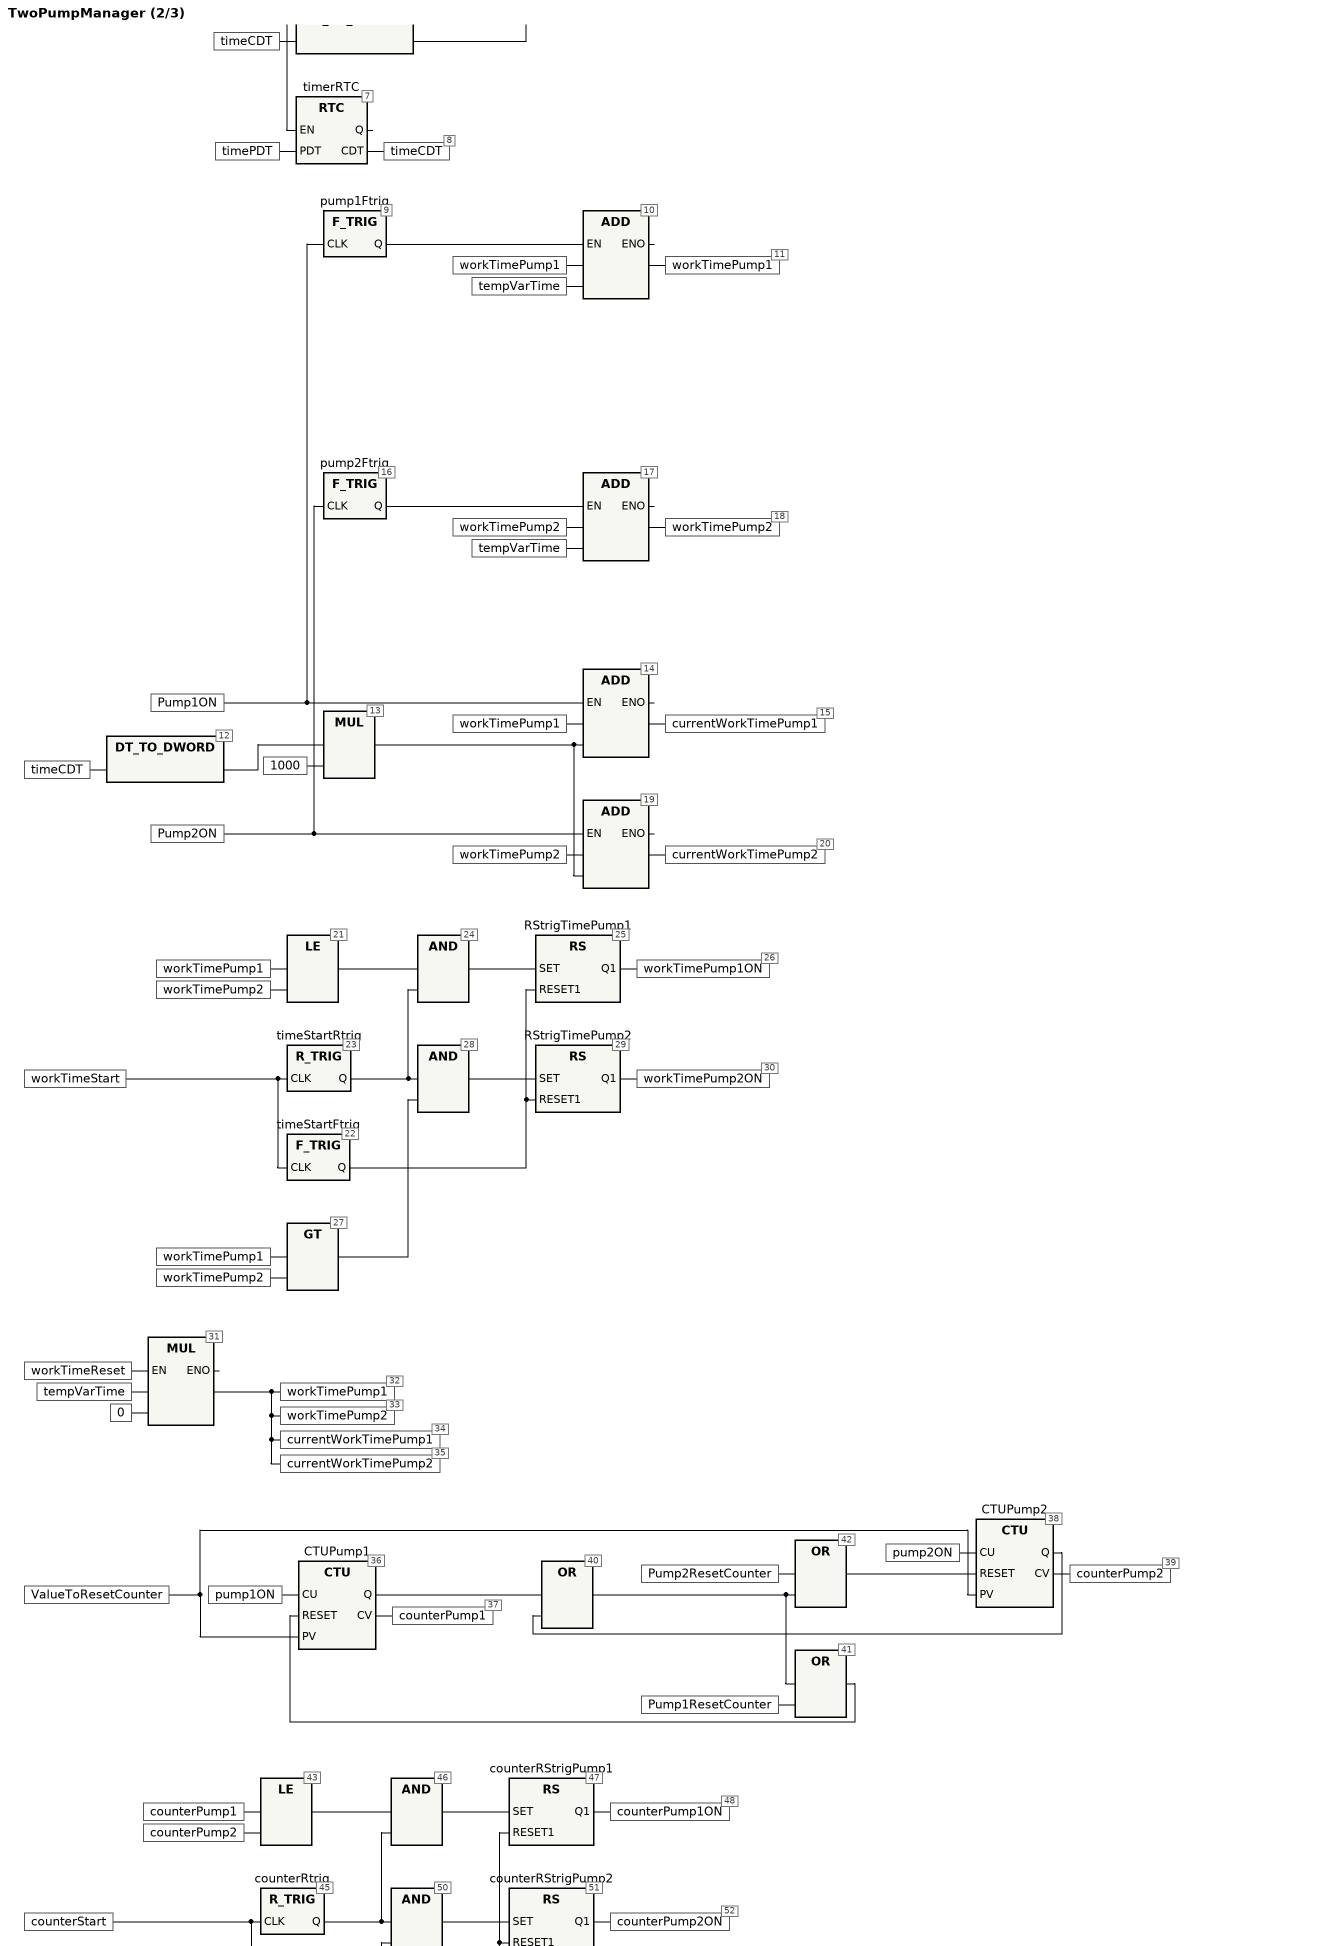
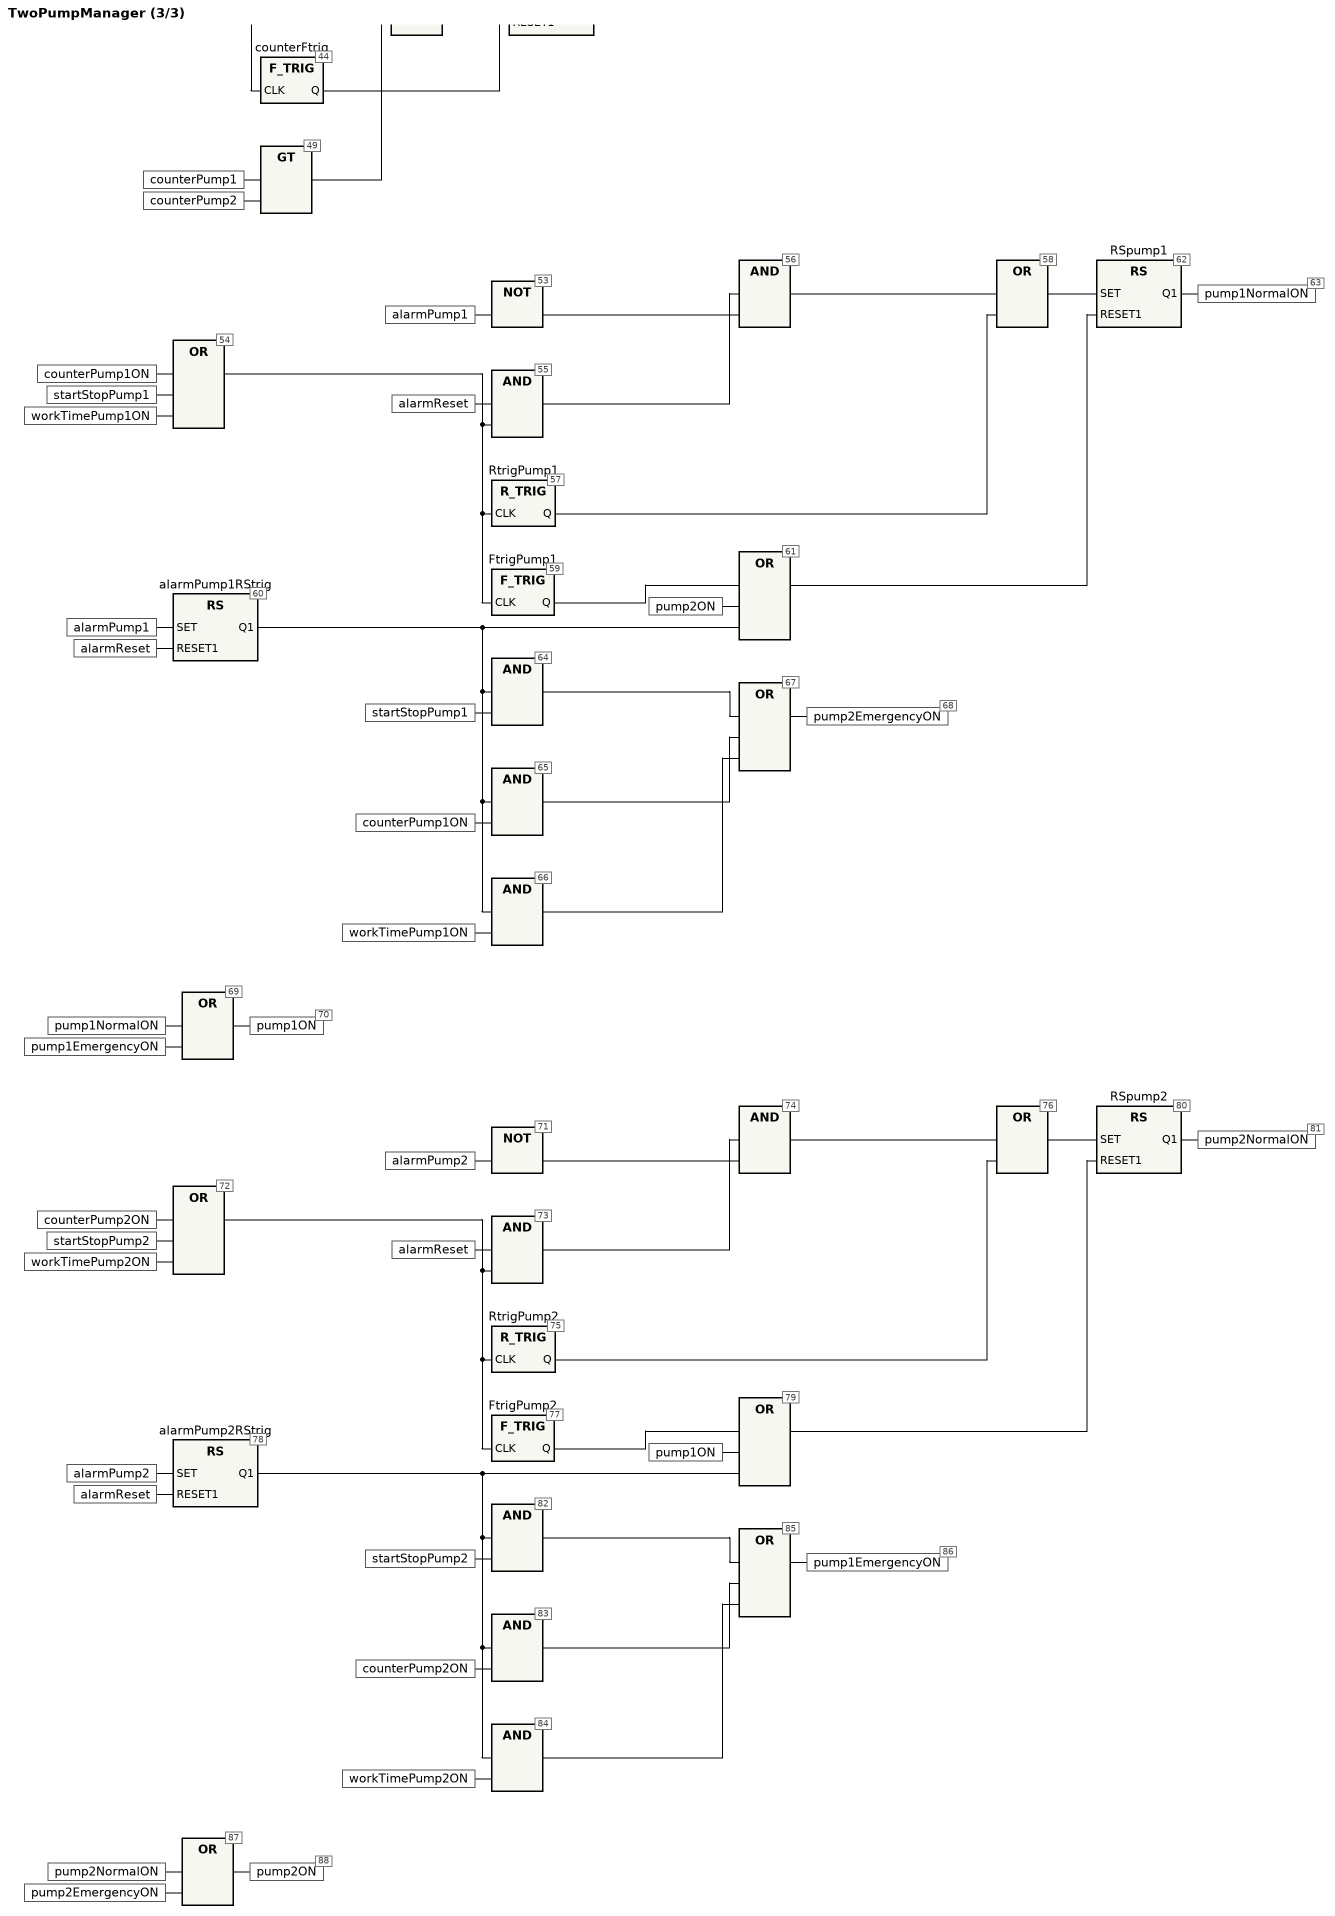
_CFC_ (* Continuous Function Chart, elements in execution order *)
(* Сброс времени наработки. *)
(* Запуск насоса с наименьшей наработкой. *)
(* Блок запуска насоса с наименьшей наработкой. / Также считает наработку насосов независимо от варианта выбора запуска. *)
(* Запуск насоса с выбором по наработке. *)
(* Если workTimePump1 <= / workTimePump2, то TRUE *)
(* Если workTimePump1 > / workTimePump2, то TRUE *)
(* Часы, при наличии неинициализированной переменной / на входе PDT отсчитывают время от 1970.01.01 (Это ноль). *)
(* Приведение к TIME *)
(* Счетчик времени наработки включенного насоса. *)
(* Выбор и запуск насоса с меньшим временем наработки *)
(* Промежуточная переменная хранения / времени наработки за включение. *)
(* Запись времени наработки первого насоса *)
(* Отображение текущей наработки первого насоса *)
(* Запись времени наработки второго насоса *)
(* Отображение текущей наработки второго насоса *)
(* Приведение к TIME *)
(* Блок управления запуском насосов с учетом количества включений. / При активации counterStart запустится насос с меньшим количеством включений. / При достижении счетчиком заданного значения ValueToResetCounter оба счетчика сбрасываются. / Если ко входу блока не подключена переменная для задания ValueToResetCounter, то сброс при достижении максимального значения переменной: 65535. *)
(* Оба счетчика сбрасываются в ноль, если хоть один достигнет заданного значения (по умолчанию 65535). *)
(* пуск/стоп pump2 по кол.вкл *)
(* пуск/стоп pump1 по кол.вкл *)
(* Если counterPump1 <= / counterPump2, то TRUE *)
(* выход на запуск второго насоса *)
(* запуск первого насоса при аварии второго *)
(* Если запущен первый насос, второй не включается *)
(* авария на втором насосе *)
(* ручной норм.пуск/стоп pump2 *)
(* выход на запуск первого насоса *)
(* ручной норм.пуск/стоп pump1 *)
(* запуск второго насоса при аварии первого *)
(* Если запущен второй насос, первый не включается *)
(* авария на первом насосе *)
(* Если был запущен первый насос, произошла его авария, включился второй насос, / а потом авария первого насоса ушла, сделали сброс аварии, то снова запустится первый насос. *)
(* второй насос включается в нормальном или аварийном режимах. *)
(* первый насос включается в нормальном или аварийном режимах. *)
(* Если был запущен второй насос, произошла его авария, включился первый насос, / а потом авария второго насоса ушла, сделали сброс аварии, то снова запустится второй насос. *)
(* Если counterPump1 > / counterPump2, то TRUE *)
(* Блок ручного управления парой насосов, которые не работают одновременно. / При аварии запущенного насоса переходит на резервный (незапущенный) насос. / Не разрешает одновременный запуск двух насосов. *)
(* пуск/стоп pump1 по наработке *)
(* пуск/стоп pump2 по наработке *)
#0 OR(Pump1ON, Pump2ON)
#1 timerFtrig:F_TRIG(CLK: #0)
#2 DT_TO_DWORD(timeCDT)
#3 ADD(EN: #1.Q, #2, 0)
#4 MUL(#3, 1000)
#5 DWORD_TO_TIME(#4)
#6 tempVarTime <= #5
#7 timerRTC:RTC(EN: #0, PDT: timePDT)
#8 timeCDT <= #7.CDT
#9 pump1Ftrig:F_TRIG(CLK: Pump1ON)
#10 ADD(EN: #9.Q, workTimePump1, tempVarTime)
#11 workTimePump1 <= #10
#12 DT_TO_DWORD(timeCDT)
#13 MUL(#12, 1000)
#14 ADD(EN: Pump1ON, workTimePump1, #13)
#15 currentWorkTimePump1 <= #14
#16 pump2Ftrig:F_TRIG(CLK: Pump2ON)
#17 ADD(EN: #16.Q, workTimePump2, tempVarTime)
#18 workTimePump2 <= #17
#19 ADD(EN: Pump2ON, workTimePump2, #13)
#20 currentWorkTimePump2 <= #19
#21 LE(workTimePump1, workTimePump2)
#22 timeStartFtrig:F_TRIG(CLK: workTimeStart)
#23 timeStartRtrig:R_TRIG(CLK: workTimeStart)
#24 AND(#21, #23.Q)
#25 RStrigTimePump1:RS(SET: #24, RESET1: #22.Q)
#26 workTimePump1ON <= #25.Q1
#27 GT(workTimePump1, workTimePump2)
#28 AND(#23.Q, #27)
#29 RStrigTimePump2:RS(SET: #28, RESET1: #22.Q)
#30 workTimePump2ON <= #29.Q1
#31 MUL(EN: workTimeReset, tempVarTime, 0)
#32 workTimePump1 <= #31
#33 workTimePump2 <= #31
#34 currentWorkTimePump1 <= #31
#35 currentWorkTimePump2 <= #31
#36 CTUPump1:CTU(CU: pump1ON, RESET: #41, PV: ValueToResetCounter)
#37 counterPump1 <= #36.CV
#38 CTUPump2:CTU(CU: pump2ON, RESET: #42, PV: ValueToResetCounter)
#39 counterPump2 <= #38.CV
#40 OR(#36.Q, #38.Q)
#41 OR(#40, Pump1ResetCounter)
#42 OR(Pump2ResetCounter, #40)
#43 LE(counterPump1, counterPump2)
#44 counterFtrig:F_TRIG(CLK: counterStart)
#45 counterRtrig:R_TRIG(CLK: counterStart)
#46 AND(#43, #45.Q)
#47 counterRStrigPump1:RS(SET: #46, RESET1: #44.Q)
#48 counterPump1ON <= #47.Q1
#49 GT(counterPump1, counterPump2)
#50 AND(#45.Q, #49)
#51 counterRStrigPump2:RS(SET: #50, RESET1: #44.Q)
#52 counterPump2ON <= #51.Q1
#53 NOT(alarmPump1)
#54 OR(counterPump1ON, startStopPump1, workTimePump1ON)
#55 AND(alarmReset, #54)
#56 AND(#55, #53)
#57 RtrigPump1:R_TRIG(CLK: #54)
#58 OR(#56, #57.Q)
#59 FtrigPump1:F_TRIG(CLK: #54)
#60 alarmPump1RStrig:RS(SET: alarmPump1, RESET1: alarmReset)
#61 OR(#59.Q, pump2ON, #60.Q1)
#62 RSpump1:RS(SET: #58, RESET1: #61)
#63 pump1NormalON <= #62.Q1
#64 AND(#60.Q1, startStopPump1)
#65 AND(#60.Q1, counterPump1ON)
#66 AND(#60.Q1, workTimePump1ON)
#67 OR(#64, #65, #66)
#68 pump2EmergencyON <= #67
#69 OR(pump1NormalON, pump1EmergencyON)
#70 pump1ON <= #69
#71 NOT(alarmPump2)
#72 OR(counterPump2ON, startStopPump2, workTimePump2ON)
#73 AND(alarmReset, #72)
#74 AND(#73, #71)
#75 RtrigPump2:R_TRIG(CLK: #72)
#76 OR(#74, #75.Q)
#77 FtrigPump2:F_TRIG(CLK: #72)
#78 alarmPump2RStrig:RS(SET: alarmPump2, RESET1: alarmReset)
#79 OR(#77.Q, pump1ON, #78.Q1)
#80 RSpump2:RS(SET: #76, RESET1: #79)
#81 pump2NormalON <= #80.Q1
#82 AND(#78.Q1, startStopPump2)
#83 AND(#78.Q1, counterPump2ON)
#84 AND(#78.Q1, workTimePump2ON)
#85 OR(#82, #83, #84)
#86 pump1EmergencyON <= #85
#87 OR(pump2NormalON, pump2EmergencyON)
#88 pump2ON <= #87
_END_CFC_
END_FUNCTION_BLOCK

(* POU DosingPumpProportional, CFC *)
FUNCTION_BLOCK DosingPumpProportional
VAR_INPUT
	flowValue: REAL;		(*текущее значение мгновенного расхода, кубометров в час.*)
	setMinPumpDosingValue: REAL := 0;		(*задание минимальной производительности доз.насоса. По умолчанию = 0.*)
	setMaxPumpDosingValue: REAL;		(*задание максимальной производительности доз.насоса, в мл/мин*)
	minOutputValue: REAL := 4;		(*минимальное значение выходного сигнала. По умолчанию = 4, сработает, если не подключать ко входу переменную.*)
	maxOutputValue: REAL := 20;		(*Максимально значение выходного сигнала. По умолчанию = 20, сработает, если не подключать ко входу переменную.*)
	setKoeffProportionality: REAL;		(*Задание мл на кубометр (коэф.пропорциональности между расходом и дозированием)*)
	minFlowToStart: REAL := 10;		(*Минимальное значение расхода для подачи сигнала на начало дозирования. По умолчанию = 10 кубометров в час, сработает, если не подключать ко входу переменную.*)
END_VAR
VAR_OUTPUT
	outputValue: REAL;		(*Выходной сигнал на дозирующий насос.*)
	startDosingPump: BOOL;		(*Сигнал на запуск дозирующего насоса.*)
	dosingError: BOOL;		(*Ошибка производительности дозирования (неверно заданы значения производительности насоса, производительность доз.насоса не соответствует расходу.*)
END_VAR
VAR
	linearTransformator: LIN_TRAFO;		(*получает на вход значение из указанного диапазона, ставит на выходе пропорциональное значение из другого диапазона.*)
END_VAR
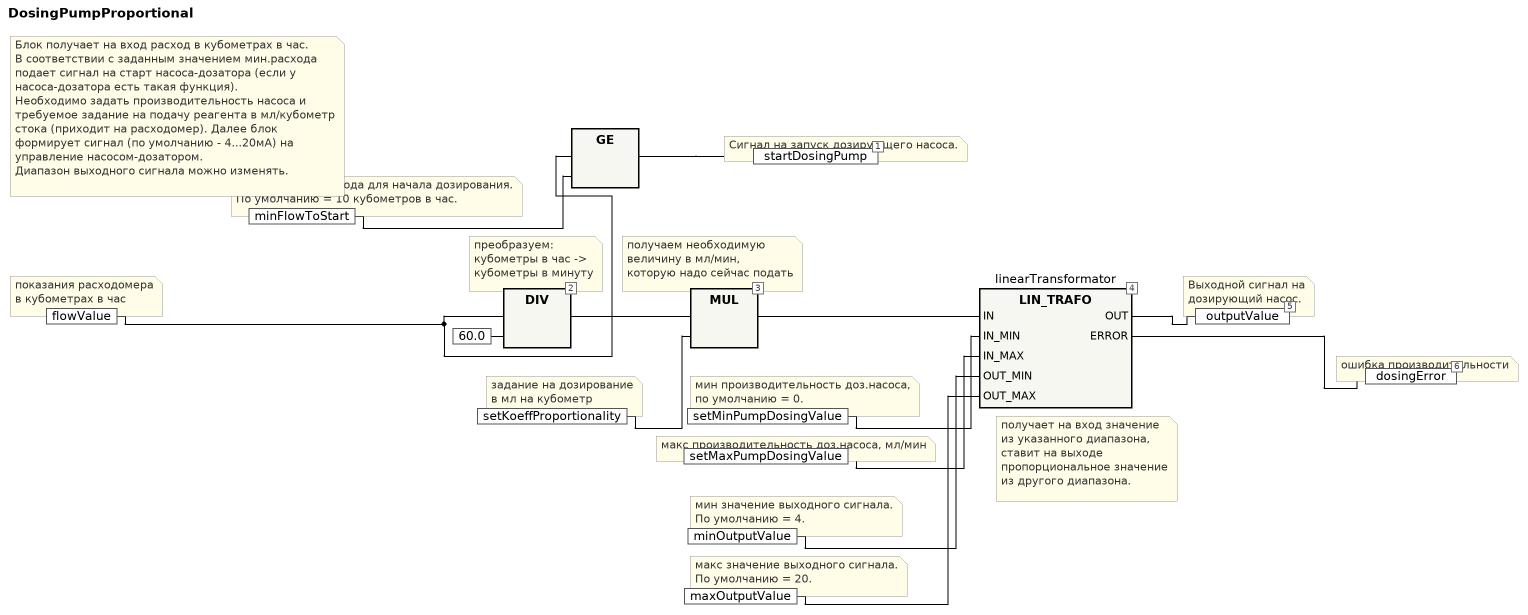
_CFC_ (* Continuous Function Chart, elements in execution order *)
(* Сигнал на запуск дозирующего насоса. *)
(* min значение расхода для начала дозирования. / По умолчанию = 10 кубометров в час. *)
(* макс производительность доз.насоса, мл/мин *)
(* мин производительность доз.насоса, / по умолчанию = 0. *)
(* получаем необходимую / величину в мл/мин, / которую надо сейчас подать *)
(* задание на дозирование / в мл на кубометр *)
(* показания расходомера / в кубометрах в час *)
(* преобразуем: / кубометры в час -> / кубометры в минуту *)
(* мин значение выходного сигнала. / По умолчанию = 4. *)
(* макс значение выходного сигнала. / По умолчанию = 20. *)
(* Выходной сигнал на / дозирующий насос. *)
(* ошибка производительности *)
(* получает на вход значение / из указанного диапазона, / ставит на выходе / пропорциональное значение / из другого диапазона. *)
(* Блок получает на вход расход в кубометрах в час. / В соответствии с заданным значением мин.расхода подает сигнал на старт насоса-дозатора (если у насоса-дозатора есть такая функция). / Необходимо задать производительность насоса и требуемое задание на подачу реагента в мл/кубометр стока (приходит на расходомер). Далее блок формирует сигнал (по умолчанию - 4...20мА) на управление насосом-дозатором. / Диапазон выходного сигнала можно изменять. *)
#0 GE(flowValue, minFlowToStart)
#1 startDosingPump <= #0
#2 DIV(flowValue, 60.0)
#3 MUL(#2, setKoeffProportionality)
#4 linearTransformator:LIN_TRAFO(IN: #3, IN_MIN: setMinPumpDosingValue, IN_MAX: setMaxPumpDosingValue, OUT_MIN: minOutputValue, OUT_MAX: maxOutputValue)
#5 outputValue <= #4.OUT
#6 dosingError <= #4.ERROR
_END_CFC_
(* the same logic as Structured Text *)
(* Сигнал на запуск дозирующего насоса. *)
(* min значение расхода для начала дозирования. / По умолчанию = 10 кубометров в час. *)
(* макс производительность доз.насоса, мл/мин *)
(* мин производительность доз.насоса, / по умолчанию = 0. *)
(* получаем необходимую / величину в мл/мин, / которую надо сейчас подать *)
(* задание на дозирование / в мл на кубометр *)
(* показания расходомера / в кубометрах в час *)
(* преобразуем: / кубометры в час -> / кубометры в минуту *)
(* мин значение выходного сигнала. / По умолчанию = 4. *)
(* макс значение выходного сигнала. / По умолчанию = 20. *)
(* Выходной сигнал на / дозирующий насос. *)
(* ошибка производительности *)
(* получает на вход значение / из указанного диапазона, / ставит на выходе / пропорциональное значение / из другого диапазона. *)
(* Блок получает на вход расход в кубометрах в час. / В соответствии с заданным значением мин.расхода подает сигнал на старт насоса-дозатора (если у насоса-дозатора есть такая функция). / Необходимо задать производительность насоса и требуемое задание на подачу реагента в мл/кубометр стока (приходит на расходомер). Далее блок формирует сигнал (по умолчанию - 4...20мА) на управление насосом-дозатором. / Диапазон выходного сигнала можно изменять. *)
startDosingPump := flowValue >= minFlowToStart;
linearTransformator(IN := (flowValue / 60.0) * setKoeffProportionality, IN_MIN := setMinPumpDosingValue, IN_MAX := setMaxPumpDosingValue, OUT_MIN := minOutputValue, OUT_MAX := maxOutputValue);
outputValue := linearTransformator.OUT;
dosingError := linearTransformator.ERROR;
END_FUNCTION_BLOCK

(* POU SimpleValve, CFC *)
FUNCTION_BLOCK SimpleValve
VAR_INPUT
	inputOpen: BOOL;		(*вход подающий сигнал на открытие*)
	inputClose: BOOL;		(*вход, подающий сигнал на закрытие*)
	statusOpen: BOOL;		(*статус: заслонка/задвижка ОТКРЫТА*)
	statusClose: BOOL;		(*статус: заслонка/задвижка ЗАКРЫТА*)
	reset: BOOL;		(*ручной сброс выходов и аварий в неактивное состояние*)
	timeToOpenClose: BYTE;		(*Время в секундах на открытие/закрытие (по тех.характеристикам прибора).*)
END_VAR
VAR_OUTPUT
	outputOpen: BOOL;		(*выход на открытие задвижки/заслонки*)
	outputClose: BOOL;		(*выход на закрытие задвижки/заслонки*)
	errorToOpen: BOOL;		(*авария на открытие - задвижка не открылась за заданное время.*)
	errorToClose: BOOL;		(*авария на закрытие - задвижка не закрылась за заданное время.*)
END_VAR
VAR
	toOpenTrigger: RS;
	toCloseTrigger: RS;
	timerToOpenClose: TON;
END_VAR
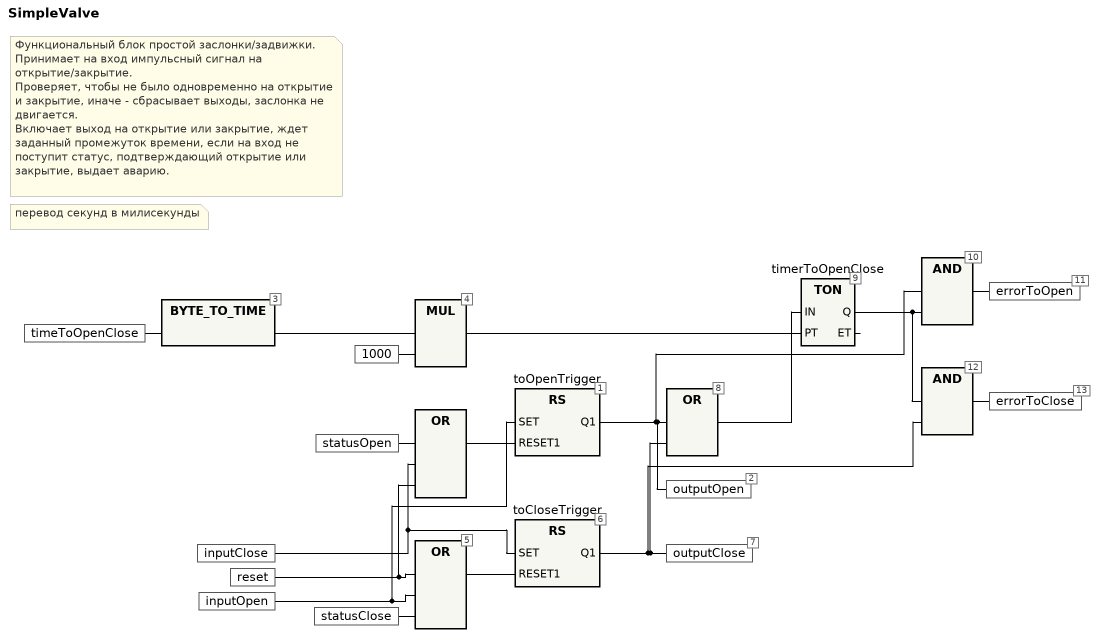
_CFC_ (* Continuous Function Chart, elements in execution order *)
(* Функциональный блок простой заслонки/задвижки. / Принимает на вход импульсный сигнал на открытие/закрытие. / Проверяет, чтобы не было одновременно на открытие и закрытие, иначе - сбрасывает выходы, заслонка не двигается. / Включает выход на открытие или закрытие, ждет заданный промежуток времени, если на вход не поступит статус, подтверждающий открытие или закрытие, выдает аварию. *)
(* перевод секунд в милисекунды *)
#0 OR(statusOpen, inputClose, reset)
#1 toOpenTrigger:RS(SET: inputOpen, RESET1: #0)
#2 outputOpen <= #1.Q1
#3 BYTE_TO_TIME(timeToOpenClose)
#4 MUL(#3, 1000)
#5 OR(reset, inputOpen, statusClose)
#6 toCloseTrigger:RS(SET: inputClose, RESET1: #5)
#7 outputClose <= #6.Q1
#8 OR(#1.Q1, #6.Q1)
#9 timerToOpenClose:TON(IN: #8, PT: #4)
#10 AND(#1.Q1, #9.Q)
#11 errorToOpen <= #10
#12 AND(#9.Q, #6.Q1)
#13 errorToClose <= #12
_END_CFC_
(* the same logic as Structured Text *)
(* Функциональный блок простой заслонки/задвижки. / Принимает на вход импульсный сигнал на открытие/закрытие. / Проверяет, чтобы не было одновременно на открытие и закрытие, иначе - сбрасывает выходы, заслонка не двигается. / Включает выход на открытие или закрытие, ждет заданный промежуток времени, если на вход не поступит статус, подтверждающий открытие или закрытие, выдает аварию. *)
(* перевод секунд в милисекунды *)
toOpenTrigger(SET := inputOpen, RESET1 := statusOpen OR inputClose OR reset);
outputOpen := toOpenTrigger.Q1;
toCloseTrigger(SET := inputClose, RESET1 := reset OR inputOpen OR statusClose);
outputClose := toCloseTrigger.Q1;
timerToOpenClose(IN := toOpenTrigger.Q1 OR toCloseTrigger.Q1, PT := BYTE_TO_TIME(timeToOpenClose) * 1000);
errorToOpen := toOpenTrigger.Q1 AND timerToOpenClose.Q;
errorToClose := timerToOpenClose.Q AND toCloseTrigger.Q1;
END_FUNCTION_BLOCK
